C01826=1195.101,-77.193,-40.224,179.414,5.586,149.159
C01827=1195.095,-76.944,-40.234,179.416,5.586,149.159
C01828=1195.090,-76.694,-40.246,179.418,5.586,149.158
C01829=1195.084,-76.444,-40.256,179.421,5.587,149.158
C01830=1195.079,-76.194,-40.267,179.423,5.587,149.157
C01831=1195.074,-75.945,-40.278,179.425,5.587,149.156
C01832=1195.068,-75.674,-40.290,179.427,5.587,149.155
C01833=1195.063,-75.403,-40.301,179.430,5.587,149.155
C01834=1195.057,-75.133,-40.313,179.433,5.588,149.154
C01835=1195.051,-74.862,-40.325,179.435,5.588,149.153
C01836=1195.046,-74.611,-40.335,179.437,5.588,149.153
C01837=1195.041,-74.362,-40.346,179.440,5.589,149.152
C01838=1195.036,-74.112,-40.357,179.442,5.589,149.151
C01839=1195.030,-73.863,-40.368,179.444,5.589,149.151
C01840=1195.025,-73.613,-40.379,179.447,5.589,149.150
C01841=1195.020,-73.363,-40.390,179.449,5.589,149.150
C01842=1195.014,-73.113,-40.401,179.451,5.589,149.149
C01843=1195.009,-72.864,-40.412,179.454,5.590,149.148
C01844=1195.004,-72.615,-40.423,179.456,5.590,149.148
C01845=1194.999,-72.364,-40.434,179.458,5.590,149.147
C01846=1194.994,-72.115,-40.445,179.460,5.590,149.146
C01847=1194.988,-71.865,-40.455,179.463,5.590,149.146
C01848=1194.983,-71.615,-40.467,179.465,5.591,149.145
C01849=1194.977,-71.366,-40.477,179.467,5.591,149.144
C01850=1194.973,-71.116,-40.489,179.470,5.591,149.144
C01851=1194.968,-70.866,-40.499,179.473,5.592,149.143
C01852=1194.962,-70.617,-40.511,179.474,5.592,149.142
C01853=1194.957,-70.367,-40.522,179.477,5.592,149.142
C01854=1194.952,-70.117,-40.533,179.479,5.592,149.141
C01855=1194.947,-69.868,-40.544,179.482,5.592,149.140
C01856=1194.941,-69.618,-40.556,179.484,5.593,149.140
C01857=1194.936,-69.368,-40.566,179.486,5.593,149.139
C01858=1194.931,-69.119,-40.577,179.489,5.593,149.138
C01859=1194.925,-68.868,-40.588,179.491,5.593,149.138
C01860=1194.921,-68.619,-40.599,179.493,5.593,149.137
C01861=1194.915,-68.370,-40.610,179.496,5.594,149.137
C01862=1194.909,-68.119,-40.622,179.498,5.594,149.136
C01863=1194.905,-67.869,-40.633,179.500,5.594,149.135
C01864=1194.900,-67.620,-40.644,179.502,5.595,149.135
C01865=1194.895,-67.370,-40.654,179.505,5.594,149.134
C01866=1194.889,-67.120,-40.666,179.507,5.595,149.133
C01867=1194.884,-66.871,-40.677,179.510,5.595,149.133
C01868=1194.879,-66.622,-40.688,179.511,5.595,149.132
C01869=1194.873,-66.371,-40.700,179.514,5.596,149.131
C01870=1194.868,-66.122,-40.711,179.517,5.596,149.131
C01871=1194.863,-65.872,-40.722,179.519,5.596,149.130
C01872=1194.858,-65.623,-40.734,179.521,5.597,149.129
C01873=1194.853,-65.372,-40.744,179.523,5.596,149.129
C01874=1194.847,-65.123,-40.756,179.526,5.597,149.128
C01875=1194.842,-64.874,-40.767,179.529,5.597,149.127
C01876=1194.838,-64.624,-40.778,179.530,5.597,149.127
C01877=1194.831,-64.374,-40.789,179.533,5.598,149.126
C01878=1194.827,-64.125,-40.801,179.535,5.598,149.125
C01879=1194.821,-63.875,-40.812,179.538,5.598,149.125
C01880=1194.816,-63.625,-40.824,179.540,5.598,149.124
C01881=1194.811,-63.375,-40.834,179.542,5.599,149.124
C01882=1194.805,-63.125,-40.846,179.544,5.598,149.123
C01883=1194.801,-62.876,-40.857,179.547,5.599,149.122
C01884=1194.795,-62.626,-40.869,179.549,5.600,149.122
C01885=1194.790,-62.377,-40.880,179.551,5.599,149.121
C01886=1194.785,-62.127,-40.891,179.554,5.600,149.120
C01887=1194.780,-61.877,-40.902,179.557,5.600,149.120
C01888=1194.775,-61.627,-40.914,179.559,5.600,149.119
C01889=1194.769,-61.378,-40.925,179.561,5.601,149.118
C01890=1194.764,-61.128,-40.936,179.563,5.600,149.118
C01891=1194.759,-60.878,-40.948,179.566,5.601,149.117
C01892=1194.754,-60.629,-40.960,179.568,5.601,149.116
C01893=1194.749,-60.379,-40.972,179.570,5.601,149.116
C01894=1194.743,-60.130,-40.982,179.573,5.602,149.115
C01895=1194.739,-59.880,-40.994,179.575,5.602,149.114
C01896=1194.733,-59.630,-41.005,179.577,5.602,149.114
C01897=1194.728,-59.380,-41.016,179.580,5.603,149.113
C01898=1194.723,-59.130,-41.028,179.582,5.603,149.112
C01899=1194.717,-58.881,-41.039,179.584,5.603,149.112
C01900=1194.712,-58.631,-41.051,179.587,5.603,149.111
C01901=1194.707,-58.382,-41.062,179.590,5.603,149.110
C01902=1194.702,-58.132,-41.074,179.591,5.604,149.110
C01903=1194.697,-57.882,-41.085,179.594,5.604,149.109
C01904=1194.691,-57.633,-41.097,179.597,5.604,149.108
C01905=1194.686,-57.383,-41.108,179.599,5.604,149.108
C01906=1194.681,-57.133,-41.120,179.601,5.605,149.107
C01907=1194.676,-56.884,-41.131,179.604,5.605,149.107
C01908=1194.671,-56.634,-41.143,179.606,5.605,149.106
C01909=1194.665,-56.384,-41.155,179.608,5.605,149.105
C01910=1194.661,-56.134,-41.166,179.611,5.606,149.104
C01911=1194.655,-55.885,-41.178,179.613,5.606,149.104
C01912=1194.650,-55.635,-41.189,179.615,5.606,149.103
C01913=1194.645,-55.385,-41.201,179.618,5.607,149.103
C01914=1194.640,-55.136,-41.212,179.620,5.606,149.102
C01915=1194.635,-54.886,-41.224,179.622,5.607,149.101
C01916=1194.630,-54.636,-41.236,179.625,5.608,149.101
C01917=1194.624,-54.386,-41.247,179.627,5.608,149.100
C01918=1194.618,-54.137,-41.259,179.630,5.608,149.099
C01919=1194.614,-53.887,-41.270,179.632,5.609,149.099
C01920=1194.609,-53.638,-41.283,179.634,5.609,149.098
C01921=1194.604,-53.388,-41.294,179.636,5.609,149.097
C01922=1194.598,-53.139,-41.306,179.639,5.609,149.097
C01923=1194.593,-52.889,-41.318,179.642,5.609,149.096
C01924=1194.588,-52.639,-41.329,179.643,5.609,149.096
C01925=1194.583,-52.389,-41.341,179.646,5.610,149.095
C01926=1194.577,-52.139,-41.353,179.649,5.610,149.094
C01927=1194.572,-51.890,-41.364,179.651,5.610,149.093
C01928=1194.567,-51.641,-41.376,179.653,5.611,149.093
C01929=1194.562,-51.391,-41.388,179.656,5.611,149.092
C01930=1194.557,-51.141,-41.400,179.658,5.611,149.092
C01931=1194.551,-50.891,-41.412,179.660,5.611,149.091
C01932=1194.547,-50.642,-41.423,179.663,5.612,149.090
C01933=1194.541,-50.392,-41.435,179.665,5.613,149.090
C01934=1194.536,-50.142,-41.447,179.667,5.612,149.089
C01935=1194.531,-49.893,-41.459,179.670,5.613,149.088
C01936=1194.525,-49.623,-41.472,179.673,5.613,149.088
C01937=1194.520,-49.353,-41.485,179.675,5.614,149.087
C01938=1194.514,-49.082,-41.497,179.677,5.613,149.086
C01939=1194.508,-48.812,-41.510,179.680,5.614,149.085
C01940=1194.504,-48.563,-41.522,179.683,5.614,149.085
C01941=1194.498,-48.313,-41.534,179.685,5.615,149.084
C01942=1194.493,-48.063,-41.545,179.687,5.615,149.084
C01943=1194.487,-47.813,-41.557,179.690,5.615,149.083
C01944=1194.483,-47.564,-41.569,179.692,5.615,149.082
C01945=1194.478,-47.314,-41.581,179.695,5.616,149.081
C01946=1194.472,-47.064,-41.593,179.697,5.616,149.081
C01947=1194.467,-46.814,-41.605,179.699,5.616,149.080
C01948=1194.462,-46.565,-41.617,179.702,5.617,149.080
C01949=1194.457,-46.315,-41.629,179.704,5.616,149.079
C01950=1194.451,-46.065,-41.641,179.707,5.617,149.078
C01951=1194.446,-45.816,-41.653,179.709,5.618,149.078
C01952=1194.442,-45.566,-41.665,179.711,5.617,149.077
C01953=1194.436,-45.316,-41.676,179.714,5.618,149.076
C01954=1194.431,-45.067,-41.689,179.716,5.618,149.076
C01955=1194.426,-44.817,-41.701,179.719,5.619,149.075
C01956=1194.420,-44.567,-41.713,179.721,5.619,149.074
C01957=1194.416,-44.318,-41.725,179.723,5.619,149.074
C01958=1194.410,-44.068,-41.737,179.726,5.620,149.073
C01959=1194.405,-43.819,-41.749,179.729,5.620,149.072
C01960=1194.400,-43.569,-41.761,179.731,5.620,149.072
C01961=1194.394,-43.319,-41.773,179.733,5.621,149.071
C01962=1194.389,-43.070,-41.786,179.735,5.621,149.070
C01963=1194.385,-42.820,-41.797,179.738,5.621,149.070
C01964=1194.379,-42.571,-41.810,179.740,5.621,149.069
C01965=1194.374,-42.321,-41.822,179.742,5.622,149.069
C01966=1194.369,-42.071,-41.833,179.745,5.622,149.068
C01967=1194.364,-41.822,-41.846,179.747,5.622,149.067
C01968=1194.358,-41.572,-41.858,179.750,5.623,149.066
C01969=1194.354,-41.323,-41.870,179.752,5.623,149.066
C01970=1194.348,-41.073,-41.882,179.755,5.624,149.065
C01971=1194.343,-40.824,-41.894,179.757,5.623,149.065
C01972=1194.338,-40.574,-41.906,179.759,5.624,149.064
C01973=1194.333,-40.324,-41.919,179.762,5.624,149.063
C01974=1194.328,-40.074,-41.931,179.764,5.624,149.062
C01975=1194.323,-39.824,-41.944,179.766,5.625,149.062
C01976=1194.317,-39.574,-41.956,179.769,5.625,149.061
C01977=1194.312,-39.325,-41.968,179.772,5.626,149.061
C01978=1194.307,-39.075,-41.980,179.774,5.625,149.060
C01979=1194.302,-38.826,-41.992,179.776,5.626,149.059
C01980=1194.297,-38.576,-42.004,179.779,5.627,149.059
C01981=1194.292,-38.327,-42.017,179.781,5.627,149.058
C01982=1194.286,-38.077,-42.028,179.783,5.627,149.057
C01983=1194.281,-37.828,-42.041,179.786,5.627,149.057
C01984=1194.276,-37.578,-42.053,179.789,5.628,149.056
C01985=1194.271,-37.328,-42.066,179.791,5.629,149.055
C01986=1194.266,-37.078,-42.078,179.793,5.628,149.055
C01987=1194.261,-36.828,-42.090,179.796,5.629,149.054
C01988=1194.256,-36.579,-42.103,179.798,5.629,149.053
C01989=1194.250,-36.329,-42.115,179.800,5.630,149.053
C01990=1194.245,-36.080,-42.127,179.802,5.630,149.052
C01991=1194.240,-35.830,-42.139,179.805,5.630,149.051
C01992=1194.234,-35.581,-42.152,179.808,5.630,149.051
C01993=1194.229,-35.331,-42.165,179.810,5.631,149.050
C01994=1194.224,-35.081,-42.177,179.812,5.631,149.050
C01995=1194.219,-34.831,-42.189,179.815,5.631,149.049
C01996=1194.214,-34.582,-42.202,179.817,5.632,149.048
C01997=1194.209,-34.332,-42.214,179.820,5.632,149.048
C01998=1194.204,-34.083,-42.226,179.822,5.632,149.047
C01999=1194.199,-33.833,-42.239,179.824,5.633,149.046
C02000=1194.193,-33.583,-42.251,179.827,5.633,149.046
C02001=1194.189,-33.333,-42.264,179.830,5.634,149.045
C02002=1194.183,-33.084,-42.277,179.832,5.633,149.044
C02003=1194.178,-32.834,-42.288,179.834,5.634,149.044
C02004=1194.173,-32.585,-42.301,179.836,5.635,149.043
C02005=1194.168,-32.336,-42.314,179.839,5.635,149.042
C02006=1194.163,-32.086,-42.327,179.842,5.636,149.042
C02007=1194.157,-31.835,-42.339,179.844,5.635,149.041
C02008=1194.152,-31.586,-42.352,179.847,5.636,149.040
C02009=1194.147,-31.337,-42.364,179.849,5.637,149.040
C02010=1194.142,-31.087,-42.377,179.851,5.637,149.039
C02011=1194.136,-30.837,-42.389,179.853,5.637,149.038
C02012=1194.132,-30.587,-42.402,179.856,5.637,149.038
C02013=1194.127,-30.338,-42.414,179.859,5.638,149.037
C02014=1194.122,-30.089,-42.427,179.861,5.638,149.037
C02015=1194.116,-29.839,-42.440,179.863,5.638,149.036
C02016=1194.112,-29.589,-42.452,179.866,5.639,149.035
C02017=1194.106,-29.339,-42.465,179.868,5.639,149.034
C02018=1194.101,-29.090,-42.478,179.871,5.639,149.034
C02019=1194.095,-28.841,-42.490,179.873,5.640,149.033
C02020=1194.090,-28.591,-42.503,179.875,5.640,149.033
C02021=1194.086,-28.341,-42.516,179.878,5.640,149.032
C02022=1194.080,-28.091,-42.528,179.881,5.641,149.031
C02023=1194.075,-27.842,-42.540,179.883,5.641,149.031
C02024=1194.069,-27.592,-42.553,179.885,5.642,149.030
C02025=1194.065,-27.342,-42.566,179.888,5.642,149.029
C02026=1194.060,-27.093,-42.579,179.890,5.642,149.029
C02027=1194.055,-26.844,-42.592,179.893,5.643,149.028
C02028=1194.050,-26.594,-42.604,179.895,5.644,149.027
C02029=1194.045,-26.344,-42.617,179.897,5.643,149.027
C02030=1194.039,-26.094,-42.630,179.900,5.644,149.026
C02031=1194.034,-25.845,-42.642,179.902,5.644,149.025
C02032=1194.029,-25.595,-42.655,179.905,5.645,149.025
C02033=1194.024,-25.345,-42.668,179.907,5.645,149.024
C02034=1194.019,-25.096,-42.680,179.909,5.645,149.024
C02035=1194.013,-24.846,-42.694,179.912,5.646,149.023
C02036=1194.009,-24.596,-42.707,179.915,5.646,149.022
C02037=1194.003,-24.347,-42.719,179.917,5.647,149.021
C02038=1193.998,-24.098,-42.732,179.919,5.647,149.021
C02039=1193.993,-23.847,-42.745,179.922,5.647,149.020
C02040=1193.987,-23.578,-42.759,179.924,5.648,149.020
C02041=1193.982,-23.309,-42.772,179.927,5.648,149.019
C02042=1193.977,-23.039,-42.787,179.930,5.648,149.018
C02043=1193.971,-22.770,-42.800,179.932,5.649,149.018
C02044=1193.966,-22.519,-42.813,179.935,5.649,149.017
C02045=1193.961,-22.270,-42.826,179.938,5.650,149.016
C02046=1193.956,-22.021,-42.839,179.940,5.650,149.015
C02047=1193.950,-21.770,-42.852,179.942,5.650,149.015
C02048=1193.946,-21.522,-42.866,179.944,5.651,149.014
C02049=1193.940,-21.272,-42.878,179.947,5.651,149.014
C02050=1193.935,-21.022,-42.892,179.950,5.652,149.013
C02051=1193.930,-20.773,-42.904,179.952,5.652,149.012
C02052=1193.925,-20.523,-42.917,179.955,5.653,149.012
C02053=1193.920,-20.273,-42.931,179.957,5.653,149.011
C02054=1193.914,-20.024,-42.943,179.959,5.653,149.010
C02055=1193.909,-19.774,-42.956,179.962,5.654,149.010
C02056=1193.904,-19.524,-42.969,179.965,5.654,149.009
C02057=1193.899,-19.275,-42.982,179.967,5.655,149.008
C02058=1193.894,-19.025,-42.995,179.969,5.655,149.008
C02059=1193.889,-18.776,-43.009,179.972,5.655,149.007
C02060=1193.884,-18.526,-43.021,179.974,5.656,149.006
C02061=1193.879,-18.276,-43.034,179.977,5.656,149.006
C02062=1193.873,-18.027,-43.048,179.979,5.657,149.005
C02063=1193.868,-17.777,-43.060,179.982,5.657,149.005
C02064=1193.863,-17.527,-43.074,179.984,5.657,149.004
C02065=1193.858,-17.278,-43.087,179.986,5.657,149.003
C02066=1193.854,-17.028,-43.100,179.989,5.658,149.002
C02067=1193.848,-16.779,-43.113,179.991,5.659,149.002
C02068=1193.843,-16.529,-43.126,179.994,5.659,149.001
C02069=1193.837,-16.279,-43.139,179.997,5.660,149.001
C02070=1193.833,-16.030,-43.153,179.999,5.659,149.000
C02071=1193.828,-15.780,-43.166,-179.999,5.660,148.999
C02072=1193.822,-15.531,-43.179,-179.997,5.661,148.999
C02073=1193.818,-15.281,-43.192,-179.994,5.661,148.998
C02074=1193.812,-15.032,-43.206,-179.991,5.662,148.997
C02075=1193.807,-14.782,-43.218,-179.989,5.662,148.997
C02076=1193.802,-14.532,-43.232,-179.986,5.663,148.996
C02077=1193.797,-14.283,-43.244,-179.984,5.663,148.995
C02078=1193.792,-14.033,-43.259,-179.982,5.663,148.995
C02079=1193.787,-13.784,-43.271,-179.979,5.664,148.994
C02080=1193.782,-13.534,-43.284,-179.976,5.664,148.993
C02081=1193.776,-13.285,-43.298,-179.974,5.665,148.993
C02082=1193.772,-13.035,-43.311,-179.972,5.665,148.992
C02083=1193.766,-12.785,-43.324,-179.969,5.665,148.992
C02084=1193.762,-12.536,-43.338,-179.967,5.666,148.991
C02085=1193.756,-12.286,-43.351,-179.964,5.666,148.990
C02086=1193.751,-12.037,-43.364,-179.962,5.667,148.990
C02087=1193.746,-11.787,-43.378,-179.959,5.667,148.989
C02088=1193.741,-11.538,-43.391,-179.957,5.668,148.988
C02089=1193.736,-11.287,-43.404,-179.954,5.668,148.988
C02090=1193.730,-11.038,-43.418,-179.952,5.668,148.987
C02091=1193.725,-10.788,-43.431,-179.950,5.669,148.986
C02092=1193.720,-10.539,-43.445,-179.947,5.669,148.986
C02093=1193.715,-10.289,-43.458,-179.944,5.670,148.985
C02094=1193.710,-10.040,-43.471,-179.942,5.670,148.984
C02095=1193.705,-9.790,-43.485,-179.939,5.671,148.984
C02096=1193.699,-9.541,-43.498,-179.937,5.672,148.983
C02097=1193.695,-9.291,-43.512,-179.935,5.671,148.983
C02098=1193.690,-9.041,-43.525,-179.932,5.672,148.982
C02099=1193.685,-8.792,-43.539,-179.930,5.672,148.981
C02100=1193.680,-8.542,-43.552,-179.927,5.673,148.980
C02101=1193.674,-8.293,-43.566,-179.925,5.674,148.980
C02102=1193.670,-8.043,-43.579,-179.922,5.674,148.979
C02103=1193.664,-7.794,-43.593,-179.919,5.674,148.979
C02104=1193.660,-7.544,-43.606,-179.917,5.675,148.978
C02105=1193.654,-7.295,-43.620,-179.915,5.675,148.977
C02106=1193.649,-7.045,-43.633,-179.913,5.675,148.977
C02107=1193.644,-6.796,-43.647,-179.910,5.676,148.976
C02108=1193.639,-6.546,-43.660,-179.907,5.676,148.975
C02109=1193.634,-6.296,-43.675,-179.905,5.677,148.975
C02110=1193.629,-6.046,-43.687,-179.902,5.678,148.974
C02111=1193.624,-5.797,-43.701,-179.900,5.678,148.974
C02112=1193.618,-5.547,-43.715,-179.897,5.679,148.973
C02113=1193.614,-5.298,-43.728,-179.894,5.679,148.972
C02114=1193.608,-5.048,-43.742,-179.892,5.679,148.971
C02115=1193.603,-4.798,-43.756,-179.890,5.680,148.971
C02116=1193.599,-4.549,-43.770,-179.888,5.680,148.970
C02117=1193.593,-4.299,-43.783,-179.885,5.681,148.970
C02118=1193.588,-4.050,-43.797,-179.882,5.681,148.969
C02119=1193.583,-3.800,-43.810,-179.880,5.682,148.969
C02120=1193.578,-3.551,-43.824,-179.877,5.682,148.968
C02121=1193.573,-3.301,-43.838,-179.875,5.683,148.967
C02122=1193.568,-3.052,-43.851,-179.872,5.683,148.966
C02123=1193.563,-2.802,-43.865,-179.870,5.683,148.966
C02124=1193.557,-2.553,-43.879,-179.868,5.684,148.965
C02125=1193.552,-2.303,-43.892,-179.865,5.684,148.965
C02126=1193.548,-2.053,-43.906,-179.863,5.685,148.964
C02127=1193.542,-1.804,-43.920,-179.860,5.685,148.963
C02128=1193.537,-1.554,-43.934,-179.857,5.686,148.963
C02129=1193.532,-1.304,-43.948,-179.855,5.687,148.962
C02130=1193.527,-1.055,-43.961,-179.852,5.687,148.961
C02131=1193.522,-0.805,-43.975,-179.850,5.688,148.961
C02132=1193.517,-0.555,-43.989,-179.847,5.688,148.960
C02133=1193.511,-0.306,-44.003,-179.845,5.689,148.960
C02134=1193.507,-0.057,-44.017,-179.843,5.689,148.959
C02135=1193.502,0.193,-44.030,-179.840,5.689,148.958
C02136=1193.496,0.442,-44.044,-179.838,5.690,148.957
C02137=1193.491,0.692,-44.058,-179.835,5.690,148.957
C02138=1193.486,0.942,-44.073,-179.833,5.691,148.956
C02139=1193.481,1.191,-44.085,-179.830,5.692,148.956
C02140=1193.476,1.441,-44.100,-179.827,5.692,148.955
C02141=1193.471,1.691,-44.114,-179.825,5.693,148.954
C02142=1193.466,1.940,-44.128,-179.823,5.693,148.954
C02143=1193.461,2.189,-44.142,-179.820,5.694,148.953
C02144=1193.455,2.459,-44.157,-179.817,5.694,148.952
C02145=1193.450,2.728,-44.172,-179.815,5.695,148.952
C02146=1193.444,2.997,-44.187,-179.812,5.695,148.951
C02147=1193.439,3.266,-44.202,-179.809,5.696,148.950
C02148=1193.434,3.516,-44.215,-179.807,5.696,148.950
C02149=1193.429,3.765,-44.230,-179.804,5.697,148.949
C02150=1193.424,4.014,-44.244,-179.801,5.697,148.948
C02151=1193.419,4.264,-44.258,-179.799,5.698,148.948
C02152=1193.414,4.514,-44.272,-179.797,5.699,148.947
C02153=1193.408,4.763,-44.286,-179.794,5.699,148.946
C02154=1193.403,5.012,-44.300,-179.792,5.699,148.946
C02155=1193.398,5.262,-44.315,-179.790,5.700,148.945
C02156=1193.393,5.513,-44.328,-179.787,5.700,148.945
C02157=1193.388,5.761,-44.341,-179.784,5.701,148.944
C02158=1193.383,6.011,-44.356,-179.782,5.701,148.943
C02159=1193.378,6.261,-44.370,-179.779,5.702,148.943
C02160=1193.374,6.510,-44.384,-179.777,5.702,148.942
C02161=1193.368,6.759,-44.398,-179.774,5.703,148.941
C02162=1193.363,7.009,-44.412,-179.772,5.703,148.941
C02163=1193.358,7.259,-44.427,-179.769,5.704,148.940
C02164=1193.353,7.508,-44.441,-179.767,5.705,148.940
C02165=1193.348,7.758,-44.455,-179.764,5.705,148.939
C02166=1193.343,8.007,-44.469,-179.761,5.706,148.938
C02167=1193.338,8.257,-44.483,-179.759,5.706,148.938
C02168=1193.333,8.507,-44.498,-179.757,5.707,148.937
C02169=1193.328,8.756,-44.512,-179.754,5.708,148.936
C02170=1193.322,9.005,-44.526,-179.751,5.708,148.936
C02171=1193.317,9.255,-44.540,-179.749,5.709,148.935
C02172=1193.312,9.505,-44.554,-179.746,5.709,148.934
C02173=1193.307,9.754,-44.569,-179.744,5.709,148.934
C02174=1193.302,10.004,-44.583,-179.742,5.710,148.933
C02175=1193.297,10.254,-44.597,-179.739,5.710,148.933
C02176=1193.292,10.502,-44.612,-179.737,5.711,148.932
C02177=1193.287,10.752,-44.626,-179.734,5.712,148.931
C02178=1193.282,11.002,-44.640,-179.732,5.712,148.931
C02179=1193.277,11.251,-44.655,-179.729,5.712,148.930
C02180=1193.272,11.501,-44.669,-179.726,5.713,148.929
C02181=1193.267,11.750,-44.683,-179.724,5.714,148.929
C02182=1193.262,12.000,-44.697,-179.722,5.714,148.928
C02183=1193.257,12.250,-44.712,-179.719,5.715,148.927
C02184=1193.252,12.499,-44.726,-179.716,5.715,148.927
C02185=1193.247,12.748,-44.741,-179.714,5.716,148.926
C02186=1193.242,12.998,-44.755,-179.711,5.717,148.926
C02187=1193.237,13.248,-44.769,-179.709,5.717,148.925
C02188=1193.231,13.497,-44.784,-179.706,5.718,148.924
C02189=1193.226,13.747,-44.798,-179.704,5.718,148.924
C02190=1193.221,13.997,-44.812,-179.701,5.719,148.923
C02191=1193.216,14.246,-44.827,-179.699,5.720,148.922
C02192=1193.212,14.495,-44.842,-179.696,5.720,148.922
C02193=1193.207,14.745,-44.856,-179.693,5.721,148.921
C02194=1193.202,14.995,-44.870,-179.691,5.721,148.921
C02195=1193.197,15.244,-44.885,-179.689,5.722,148.920
C02196=1193.191,15.493,-44.900,-179.686,5.722,148.919
C02197=1193.186,15.743,-44.914,-179.683,5.723,148.919
C02198=1193.181,15.993,-44.928,-179.681,5.724,148.918
C02199=1193.176,16.242,-44.943,-179.679,5.724,148.917
C02200=1193.171,16.491,-44.958,-179.676,5.725,148.917
C02201=1193.166,16.741,-44.972,-179.673,5.725,148.916
C02202=1193.161,16.990,-44.987,-179.671,5.726,148.916
C02203=1193.156,17.240,-45.002,-179.668,5.727,148.915
C02204=1193.151,17.490,-45.016,-179.666,5.727,148.914
C02205=1193.146,17.740,-45.030,-179.663,5.728,148.914
C02206=1193.141,17.989,-45.045,-179.661,5.728,148.913
C02207=1193.136,18.238,-45.060,-179.658,5.729,148.912
C02208=1193.131,18.488,-45.074,-179.656,5.729,148.912
C02209=1193.126,18.738,-45.089,-179.653,5.730,148.911
C02210=1193.120,18.987,-45.103,-179.651,5.731,148.911
C02211=1193.116,19.236,-45.118,-179.648,5.731,148.910
C02212=1193.110,19.486,-45.133,-179.646,5.732,148.909
C02213=1193.105,19.735,-45.147,-179.643,5.732,148.909
C02214=1193.101,19.984,-45.162,-179.641,5.733,148.908
C02215=1193.096,20.234,-45.177,-179.638,5.734,148.907
C02216=1193.090,20.484,-45.192,-179.635,5.734,148.907
C02217=1193.085,20.733,-45.207,-179.633,5.735,148.906
C02218=1193.080,20.983,-45.221,-179.631,5.736,148.906
C02219=1193.076,21.232,-45.236,-179.628,5.736,148.905
C02220=1193.070,21.482,-45.251,-179.625,5.737,148.904
C02221=1193.065,21.731,-45.266,-179.623,5.737,148.904
C02222=1193.060,21.981,-45.280,-179.621,5.738,148.903
C02223=1193.055,22.230,-45.296,-179.618,5.738,148.902
C02224=1193.050,22.480,-45.310,-179.615,5.739,148.902
C02225=1193.045,22.729,-45.325,-179.613,5.739,148.901
C02226=1193.040,22.979,-45.339,-179.610,5.740,148.901
C02227=1193.035,23.228,-45.355,-179.608,5.741,148.900
C02228=1193.030,23.478,-45.369,-179.605,5.741,148.899
C02229=1193.025,23.727,-45.384,-179.602,5.742,148.899
C02230=1193.020,23.977,-45.399,-179.600,5.743,148.898
C02231=1193.015,24.226,-45.414,-179.598,5.743,148.897
C02232=1193.010,24.476,-45.428,-179.595,5.744,148.897
C02233=1193.005,24.725,-45.444,-179.592,5.744,148.896
C02234=1193.000,24.975,-45.458,-179.590,5.745,148.896
C02235=1192.994,25.224,-45.474,-179.588,5.746,148.895
C02236=1192.990,25.474,-45.489,-179.585,5.746,148.894
C02237=1192.985,25.724,-45.503,-179.583,5.747,148.894
C02238=1192.980,25.973,-45.519,-179.580,5.748,148.893
C02239=1192.975,26.223,-45.533,-179.577,5.748,148.893
C02240=1192.970,26.472,-45.549,-179.574,5.749,148.892
C02241=1192.965,26.721,-45.564,-179.572,5.750,148.891
C02242=1192.960,26.971,-45.578,-179.569,5.751,148.891
C02243=1192.955,27.221,-45.594,-179.567,5.751,148.890
C02244=1192.950,27.470,-45.608,-179.564,5.752,148.889
C02245=1192.944,27.720,-45.623,-179.562,5.753,148.889
C02246=1192.940,27.969,-45.638,-179.559,5.753,148.888
C02247=1192.935,28.218,-45.653,-179.557,5.754,148.888
C02248=1192.929,28.487,-45.670,-179.554,5.754,148.887
C02249=1192.923,28.756,-45.686,-179.551,5.755,148.886
C02250=1192.918,29.025,-45.702,-179.548,5.756,148.886
C02251=1192.913,29.293,-45.719,-179.546,5.756,148.885
C02252=1192.908,29.542,-45.734,-179.543,5.757,148.884
C02253=1192.903,29.793,-45.749,-179.541,5.758,148.884
C02254=1192.898,30.042,-45.764,-179.538,5.758,148.883
C02255=1192.893,30.292,-45.779,-179.536,5.759,148.883
C02256=1192.888,30.541,-45.794,-179.533,5.760,148.882
C02257=1192.882,30.791,-45.809,-179.531,5.760,148.881
C02258=1192.878,31.040,-45.824,-179.528,5.761,148.881
C02259=1192.872,31.289,-45.840,-179.526,5.762,148.880
C02260=1192.868,31.539,-45.855,-179.523,5.762,148.879
C02261=1192.863,31.789,-45.870,-179.521,5.763,148.879
C02262=1192.858,32.038,-45.885,-179.518,5.763,148.878
C02263=1192.853,32.288,-45.901,-179.515,5.765,148.878
C02264=1192.848,32.537,-45.916,-179.513,5.765,148.877
C02265=1192.843,32.786,-45.931,-179.510,5.766,148.876
C02266=1192.838,33.036,-45.946,-179.508,5.767,148.876
C02267=1192.833,33.286,-45.962,-179.505,5.767,148.875
C02268=1192.828,33.535,-45.977,-179.502,5.768,148.874
C02269=1192.823,33.784,-45.992,-179.500,5.768,148.874
C02270=1192.817,34.034,-46.008,-179.498,5.769,148.873
C02271=1192.813,34.283,-46.023,-179.495,5.770,148.873
C02272=1192.808,34.533,-46.039,-179.492,5.770,148.872
C02273=1192.803,34.782,-46.054,-179.490,5.771,148.872
C02274=1192.798,35.031,-46.069,-179.488,5.772,148.871
C02275=1192.792,35.281,-46.084,-179.484,5.773,148.870
C02276=1192.788,35.531,-46.099,-179.482,5.773,148.870
C02277=1192.783,35.781,-46.115,-179.480,5.774,148.869
C02278=1192.778,36.030,-46.130,-179.477,5.775,148.868
C02279=1192.773,36.279,-46.146,-179.474,5.775,148.868
C02280=1192.767,36.529,-46.161,-179.472,5.776,148.867
C02281=1192.763,36.778,-46.177,-179.469,5.777,148.867
C02282=1192.758,37.028,-46.192,-179.467,5.777,148.866
C02283=1192.753,37.277,-46.208,-179.464,5.778,148.865
C02284=1192.748,37.526,-46.223,-179.462,5.779,148.865
C02285=1192.743,37.776,-46.238,-179.459,5.779,148.864
C02286=1192.738,38.026,-46.254,-179.456,5.780,148.863
C02287=1192.733,38.275,-46.269,-179.454,5.781,148.863
C02288=1192.728,38.524,-46.285,-179.451,5.782,148.862
C02289=1192.722,38.774,-46.300,-179.449,5.782,148.862
C02290=1192.718,39.024,-46.316,-179.447,5.783,148.861
C02291=1192.713,39.273,-46.331,-179.444,5.784,148.861
C02292=1192.708,39.522,-46.347,-179.441,5.784,148.860
C02293=1192.703,39.772,-46.363,-179.439,5.785,148.859
C02294=1192.698,40.021,-46.378,-179.436,5.786,148.859
C02295=1192.693,40.270,-46.394,-179.433,5.787,148.858
C02296=1192.688,40.520,-46.410,-179.431,5.788,148.857
C02297=1192.683,40.770,-46.426,-179.428,5.788,148.857
C02298=1192.678,41.019,-46.441,-179.426,5.789,148.856
C02299=1192.673,41.268,-46.456,-179.423,5.789,148.856
C02300=1192.668,41.518,-46.472,-179.421,5.790,148.855
C02301=1192.663,41.768,-46.488,-179.418,5.791,148.855
C02302=1192.658,42.017,-46.503,-179.416,5.791,148.854
C02303=1192.654,42.266,-46.520,-179.413,5.793,148.853
C02304=1192.648,42.516,-46.535,-179.410,5.794,148.853
C02305=1192.643,42.765,-46.551,-179.408,5.794,148.852
C02306=1192.637,43.015,-46.566,-179.405,5.795,148.851
C02307=1192.633,43.264,-46.582,-179.403,5.796,148.851
C02308=1192.628,43.513,-46.598,-179.400,5.796,148.850
C02309=1192.623,43.763,-46.614,-179.398,5.797,148.850
C02310=1192.618,44.013,-46.630,-179.396,5.797,148.849
C02311=1192.613,44.262,-46.645,-179.392,5.799,148.848
C02312=1192.608,44.512,-46.661,-179.390,5.799,148.848
C02313=1192.604,44.761,-46.677,-179.388,5.800,148.847
C02314=1192.598,45.010,-46.692,-179.385,5.801,148.847
C02315=1192.593,45.260,-46.708,-179.382,5.801,148.846
C02316=1192.588,45.510,-46.724,-179.380,5.802,148.846
C02317=1192.583,45.758,-46.740,-179.377,5.803,148.845
C02318=1192.578,46.008,-46.756,-179.374,5.804,148.844
C02319=1192.573,46.258,-46.772,-179.372,5.805,148.844
C02320=1192.569,46.507,-46.788,-179.369,5.805,148.843
C02321=1192.564,46.756,-46.803,-179.367,5.806,148.842
C02322=1192.558,47.006,-46.819,-179.364,5.806,148.842
C02323=1192.554,47.255,-46.836,-179.362,5.807,148.841
C02324=1192.548,47.505,-46.851,-179.359,5.809,148.841
C02325=1192.544,47.755,-46.867,-179.356,5.809,148.840
C02326=1192.538,48.004,-46.884,-179.354,5.810,148.840
C02327=1192.533,48.253,-46.899,-179.351,5.811,148.839
C02328=1192.528,48.503,-46.915,-179.349,5.811,148.838
C02329=1192.523,48.752,-46.931,-179.347,5.812,148.838
C02330=1192.518,49.002,-46.947,-179.343,5.813,148.837
C02331=1192.513,49.251,-46.964,-179.341,5.814,148.836
C02332=1192.508,49.500,-46.979,-179.339,5.815,148.836
C02333=1192.503,49.750,-46.995,-179.336,5.815,148.835
C02334=1192.499,49.999,-47.011,-179.333,5.816,148.835
C02335=1192.494,50.249,-47.027,-179.331,5.817,148.834
C02336=1192.489,50.498,-47.043,-179.328,5.818,148.834
C02337=1192.484,50.748,-47.059,-179.325,5.819,148.833
C02338=1192.479,50.996,-47.075,-179.323,5.819,148.832
C02339=1192.474,51.247,-47.091,-179.320,5.820,148.832
C02340=1192.469,51.495,-47.108,-179.318,5.821,148.831
C02341=1192.464,51.745,-47.124,-179.316,5.821,148.831
C02342=1192.459,51.994,-47.140,-179.312,5.823,148.830
C02343=1192.455,52.244,-47.156,-179.310,5.823,148.829
C02344=1192.450,52.493,-47.172,-179.308,5.824,148.829
C02345=1192.444,52.744,-47.189,-179.305,5.825,148.828
C02346=1192.439,52.992,-47.205,-179.302,5.825,148.828
C02347=1192.434,53.242,-47.221,-179.300,5.827,148.827
C02348=1192.429,53.491,-47.237,-179.297,5.827,148.826
C02349=1192.425,53.741,-47.254,-179.294,5.828,148.826
C02350=1192.419,53.990,-47.270,-179.292,5.829,148.825
C02351=1192.415,54.240,-47.286,-179.290,5.829,148.825
C02352=1192.409,54.508,-47.303,-179.286,5.831,148.824
C02353=1192.404,54.777,-47.320,-179.284,5.831,148.823
C02354=1192.399,55.045,-47.338,-179.282,5.832,148.823
C02355=1192.393,55.314,-47.356,-179.278,5.834,148.822
C02356=1192.388,55.563,-47.372,-179.276,5.834,148.822
C02357=1192.383,55.812,-47.389,-179.273,5.835,148.821
C02358=1192.378,56.062,-47.405,-179.271,5.835,148.820
C02359=1192.373,56.311,-47.421,-179.268,5.837,148.820
C02360=1192.368,56.561,-47.437,-179.265,5.837,148.819
C02361=1192.363,56.810,-47.453,-179.263,5.838,148.819
C02362=1192.359,57.059,-47.470,-179.260,5.839,148.818
C02363=1192.353,57.309,-47.487,-179.258,5.840,148.818
C02364=1192.348,57.559,-47.503,-179.255,5.841,148.817
C02365=1192.343,57.807,-47.519,-179.252,5.842,148.816
C02366=1192.339,58.057,-47.536,-179.250,5.842,148.816
C02367=1192.333,58.306,-47.552,-179.248,5.843,148.815
C02368=1192.329,58.556,-47.568,-179.245,5.844,148.815
C02369=1192.324,58.806,-47.585,-179.242,5.845,148.814
C02370=1192.319,59.054,-47.602,-179.240,5.846,148.813
C02371=1192.314,59.304,-47.618,-179.237,5.846,148.813
C02372=1192.309,59.553,-47.634,-179.235,5.847,148.812
C02373=1192.304,59.803,-47.651,-179.232,5.849,148.812
C02374=1192.299,60.053,-47.668,-179.229,5.849,148.811
C02375=1192.294,60.301,-47.684,-179.227,5.850,148.811
C02376=1192.289,60.551,-47.700,-179.224,5.850,148.810
C02377=1192.284,60.800,-47.717,-179.222,5.851,148.809
C02378=1192.279,61.050,-47.734,-179.219,5.853,148.809
C02379=1192.274,61.299,-47.750,-179.216,5.853,148.808
C02380=1192.269,61.548,-47.767,-179.214,5.854,148.808
C02381=1192.265,61.798,-47.783,-179.211,5.855,148.807
C02382=1192.259,62.048,-47.800,-179.208,5.856,148.806
C02383=1192.254,62.297,-47.816,-179.206,5.857,148.806
C02384=1192.250,62.546,-47.833,-179.203,5.857,148.805
C02385=1192.244,62.796,-47.850,-179.201,5.858,148.805
C02386=1192.239,63.045,-47.867,-179.198,5.860,148.804
C02387=1192.235,63.294,-47.883,-179.195,5.860,148.804
C02388=1192.230,63.544,-47.900,-179.193,5.861,148.803
C02389=1192.225,63.793,-47.917,-179.191,5.862,148.802
C02390=1192.220,64.043,-47.933,-179.187,5.863,148.802
C02391=1192.216,64.292,-47.950,-179.185,5.864,148.801
C02392=1192.210,64.541,-47.967,-179.183,5.864,148.801
C02393=1192.205,64.791,-47.984,-179.181,5.865,148.800
C02394=1192.201,65.040,-48.000,-179.177,5.867,148.800
C02395=1192.195,65.289,-48.017,-179.175,5.867,148.799
C02396=1192.190,65.539,-48.033,-179.173,5.868,148.798
C02397=1192.185,65.789,-48.050,-179.170,5.869,148.798
C02398=1192.180,66.037,-48.067,-179.167,5.870,148.797
C02399=1192.176,66.287,-48.084,-179.165,5.871,148.797
C02400=1192.171,66.537,-48.101,-179.162,5.872,148.796
C02401=1192.166,66.786,-48.118,-179.160,5.872,148.796
C02402=1192.161,67.035,-48.134,-179.157,5.874,148.795
C02403=1192.156,67.285,-48.152,-179.154,5.875,148.795
C02404=1192.151,67.534,-48.168,-179.152,5.875,148.794
C02405=1192.145,67.783,-48.185,-179.149,5.877,148.793
C02406=1192.141,68.033,-48.202,-179.146,5.877,148.793
C02407=1192.136,68.282,-48.219,-179.144,5.878,148.792
C02408=1192.131,68.532,-48.236,-179.142,5.879,148.792
C02409=1192.126,68.781,-48.252,-179.138,5.880,148.791
C02410=1192.121,69.030,-48.269,-179.136,5.881,148.790
C02411=1192.117,69.280,-48.286,-179.134,5.882,148.790
C02412=1192.112,69.529,-48.304,-179.131,5.882,148.789
C02413=1192.107,69.779,-48.321,-179.128,5.884,148.789
C02414=1192.101,70.028,-48.338,-179.126,5.885,148.788
C02415=1192.097,70.277,-48.354,-179.123,5.885,148.788
C02416=1192.092,70.527,-48.372,-179.120,5.887,148.787
C02417=1192.087,70.777,-48.388,-179.118,5.887,148.786
C02418=1192.082,71.025,-48.406,-179.116,5.888,148.786
C02419=1192.077,71.274,-48.422,-179.113,5.889,148.785
C02420=1192.072,71.524,-48.440,-179.110,5.890,148.785
C02421=1192.067,71.774,-48.456,-179.108,5.891,148.784
C02422=1192.063,72.023,-48.474,-179.105,5.892,148.784
C02423=1192.057,72.272,-48.491,-179.102,5.893,148.783
C02424=1192.052,72.521,-48.508,-179.100,5.894,148.783
C02425=1192.048,72.771,-48.525,-179.097,5.894,148.782
C02426=1192.043,73.020,-48.543,-179.094,5.896,148.781
C02427=1192.038,73.270,-48.559,-179.092,5.897,148.781
C02428=1192.033,73.519,-48.577,-179.089,5.898,148.780
C02429=1192.027,73.769,-48.593,-179.087,5.898,148.780
C02430=1192.023,74.017,-48.611,-179.084,5.900,148.779
C02431=1192.018,74.267,-48.628,-179.081,5.900,148.779
C02432=1192.013,74.517,-48.645,-179.079,5.901,148.778
C02433=1192.009,74.766,-48.663,-179.076,5.903,148.778
C02434=1192.003,75.016,-48.680,-179.074,5.903,148.777
C02435=1191.998,75.264,-48.696,-179.071,5.904,148.776
C02436=1191.993,75.514,-48.714,-179.068,5.905,148.776
C02437=1191.989,75.763,-48.731,-179.066,5.906,148.775
C02438=1191.984,76.013,-48.748,-179.063,5.907,148.775
C02439=1191.979,76.262,-48.766,-179.060,5.908,148.774
C02440=1191.974,76.512,-48.783,-179.058,5.909,148.774
C02441=1191.969,76.761,-48.801,-179.055,5.910,148.773
C02442=1191.964,77.011,-48.818,-179.053,5.911,148.773
C02443=1191.959,77.259,-48.834,-179.050,5.912,148.772
C02444=1191.954,77.508,-48.852,-179.048,5.913,148.771
C02445=1191.949,77.758,-48.870,-179.045,5.914,148.771
C02446=1191.945,78.007,-48.887,-179.042,5.915,148.770
C02447=1191.940,78.257,-48.904,-179.040,5.916,148.770
C02448=1191.935,78.506,-48.922,-179.037,5.917,148.769
C02449=1191.930,78.756,-48.939,-179.035,5.918,148.769
C02450=1191.925,79.005,-48.957,-179.032,5.919,148.768
C02451=1191.920,79.255,-48.974,-179.029,5.920,148.768
C02452=1191.915,79.504,-48.992,-179.027,5.921,148.767
C02453=1191.911,79.753,-49.009,-179.024,5.921,148.766
C02454=1191.906,80.002,-49.027,-179.021,5.923,148.766
C02455=1191.900,80.251,-49.044,-179.019,5.924,148.765
C02456=1191.895,80.520,-49.063,-179.017,5.925,148.765
C02457=1191.890,80.788,-49.081,-179.013,5.926,148.764
C02458=1191.885,81.057,-49.101,-179.010,5.927,148.763
C02459=1191.880,81.325,-49.119,-179.008,5.928,148.763
C02460=1191.875,81.575,-49.137,-179.005,5.929,148.762
C02461=1191.869,81.824,-49.154,-179.002,5.930,148.762
C02462=1191.865,82.073,-49.172,-179.000,5.931,148.761
C02463=1191.860,82.322,-49.189,-178.997,5.932,148.761
C02464=1191.855,82.572,-49.207,-178.995,5.933,148.760
C02465=1191.850,82.821,-49.225,-178.992,5.934,148.760
C02466=1191.844,83.070,-49.242,-178.989,5.936,148.759
C02467=1191.840,83.319,-49.259,-178.987,5.936,148.758
C02468=1191.835,83.569,-49.277,-178.985,5.937,148.758
C02469=1191.830,83.818,-49.295,-178.981,5.938,148.757
C02470=1191.825,84.067,-49.313,-178.979,5.939,148.757
C02471=1191.820,84.317,-49.331,-178.977,5.940,148.756
C02472=1191.815,84.566,-49.348,-178.973,5.941,148.756
C02473=1191.811,84.815,-49.365,-178.971,5.942,148.755
C02474=1191.806,85.065,-49.383,-178.968,5.943,148.755
C02475=1191.801,85.314,-49.401,-178.966,5.944,148.754
C02476=1191.797,85.564,-49.419,-178.963,5.945,148.754
C02477=1191.792,85.813,-49.437,-178.961,5.947,148.753
C02478=1191.787,86.063,-49.455,-178.958,5.947,148.752
C02479=1191.782,86.312,-49.473,-178.956,5.948,148.752
C02480=1191.777,86.562,-49.490,-178.953,5.950,148.751
C02481=1191.772,86.811,-49.508,-178.951,5.950,148.751
C02482=1191.767,87.060,-49.525,-178.947,5.952,148.750
C02483=1191.763,87.309,-49.543,-178.945,5.953,148.750
C02484=1191.758,87.558,-49.561,-178.943,5.953,148.749
C02485=1191.752,87.808,-49.579,-178.940,5.955,148.749
C02486=1191.748,88.057,-49.597,-178.937,5.956,148.748
C02487=1191.743,88.306,-49.615,-178.934,5.957,148.748
C02488=1191.738,88.555,-49.633,-178.932,5.958,148.747
C02489=1191.733,88.804,-49.651,-178.929,5.958,148.746
C02490=1191.728,89.054,-49.669,-178.927,5.960,148.746
C02491=1191.723,89.303,-49.686,-178.924,5.961,148.745
C02492=1191.718,89.553,-49.704,-178.921,5.962,148.745
C02493=1191.713,89.802,-49.722,-178.919,5.963,148.744
C02494=1191.709,90.052,-49.740,-178.916,5.964,148.744
C02495=1191.704,90.301,-49.758,-178.913,5.965,148.743
C02496=1191.699,90.550,-49.776,-178.911,5.966,148.743
C02497=1191.694,90.799,-49.794,-178.908,5.968,148.742
C02498=1191.689,91.048,-49.812,-178.906,5.968,148.742
C02499=1191.684,91.297,-49.830,-178.903,5.969,148.741
C02500=1191.680,91.547,-49.848,-178.900,5.971,148.741
C02501=1191.675,91.797,-49.866,-178.898,5.971,148.740
C02502=1191.670,92.046,-49.884,-178.895,5.973,148.740
C02503=1191.665,92.295,-49.902,-178.892,5.974,148.739
C02504=1191.660,92.544,-49.920,-178.890,5.975,148.739
C02505=1191.655,92.793,-49.938,-178.887,5.976,148.738
C02506=1191.650,93.042,-49.956,-178.885,5.977,148.738
C02507=1191.645,93.293,-49.975,-178.882,5.978,148.737
C02508=1191.640,93.542,-49.993,-178.880,5.979,148.736
C02509=1191.635,93.791,-50.011,-178.876,5.981,148.736
C02510=1191.630,94.040,-50.029,-178.874,5.981,148.735
C02511=1191.625,94.289,-50.047,-178.872,5.982,148.735
C02512=1191.621,94.538,-50.065,-178.869,5.984,148.734
C02513=1191.616,94.788,-50.083,-178.867,5.985,148.734
C02514=1191.611,95.038,-50.101,-178.864,5.986,148.733
C02515=1191.606,95.287,-50.119,-178.862,5.987,148.733
C02516=1191.601,95.536,-50.139,-178.858,5.988,148.732
C02517=1191.596,95.785,-50.157,-178.856,5.989,148.732
C02518=1191.592,96.035,-50.175,-178.854,5.990,148.731
C02519=1191.587,96.284,-50.193,-178.851,5.992,148.731
C02520=1191.582,96.533,-50.211,-178.848,5.992,148.730
C02521=1191.577,96.782,-50.229,-178.846,5.994,148.730
C02522=1191.572,97.032,-50.248,-178.843,5.994,148.729
C02523=1191.567,97.281,-50.267,-178.840,5.996,148.729
C02524=1191.563,97.530,-50.285,-178.838,5.997,148.728
C02525=1191.558,97.779,-50.303,-178.835,5.998,148.728
C02526=1191.553,98.028,-50.321,-178.832,5.999,148.727
C02527=1191.548,98.279,-50.340,-178.830,6.001,148.726
C02528=1191.543,98.527,-50.358,-178.827,6.001,148.726
C02529=1191.538,98.776,-50.376,-178.825,6.002,148.725
C02530=1191.533,99.026,-50.394,-178.822,6.004,148.725
C02531=1191.529,99.275,-50.413,-178.820,6.005,148.724
C02532=1191.524,99.524,-50.432,-178.817,6.006,148.724
C02533=1191.519,99.773,-50.450,-178.814,6.007,148.723
C02534=1191.514,100.023,-50.468,-178.811,6.009,148.723
C02535=1191.510,100.272,-50.487,-178.809,6.009,148.722
C02536=1191.504,100.521,-50.505,-178.806,6.011,148.722
C02537=1191.499,100.771,-50.523,-178.804,6.011,148.721
C02538=1191.495,101.020,-50.542,-178.801,6.013,148.721
C02539=1191.490,101.269,-50.561,-178.798,6.014,148.720
C02540=1191.485,101.518,-50.579,-178.795,6.015,148.720
C02541=1191.481,101.768,-50.598,-178.793,6.016,148.719
C02542=1191.475,102.017,-50.617,-178.790,6.018,148.719
C02543=1191.470,102.266,-50.635,-178.788,6.019,148.718
C02544=1191.466,102.516,-50.654,-178.785,6.020,148.718
C02545=1191.461,102.765,-50.672,-178.783,6.021,148.717
C02546=1191.456,103.014,-50.690,-178.780,6.022,148.717
C02547=1191.452,103.264,-50.709,-178.777,6.023,148.716
C02548=1191.446,103.513,-50.728,-178.775,6.024,148.716
C02549=1191.441,103.762,-50.747,-178.772,6.026,148.715
C02550=1191.437,104.011,-50.765,-178.769,6.026,148.714
C02551=1191.432,104.260,-50.784,-178.767,6.028,148.714
C02552=1191.427,104.510,-50.802,-178.765,6.029,148.714
C02553=1191.423,104.759,-50.821,-178.761,6.030,148.713
C02554=1191.417,105.008,-50.840,-178.759,6.031,148.713
C02555=1191.412,105.257,-50.859,-178.756,6.033,148.712
C02556=1191.407,105.507,-50.877,-178.754,6.034,148.712
C02557=1191.403,105.756,-50.896,-178.751,6.035,148.711
C02558=1191.398,106.005,-50.914,-178.749,6.036,148.710
C02559=1191.393,106.254,-50.934,-178.746,6.038,148.710
C02560=1191.388,106.523,-50.953,-178.743,6.039,148.709
C02561=1191.383,106.791,-50.974,-178.740,6.040,148.709
C02562=1191.377,107.060,-50.994,-178.737,6.041,148.708
C02563=1191.372,107.328,-51.014,-178.734,6.043,148.708
C02564=1191.367,107.578,-51.033,-178.732,6.044,148.707
C02565=1191.363,107.826,-51.052,-178.729,6.045,148.707
C02566=1191.358,108.076,-51.071,-178.727,6.046,148.706
C02567=1191.353,108.325,-51.090,-178.724,6.047,148.706
C02568=1191.348,108.574,-51.108,-178.721,6.048,148.705
C02569=1191.344,108.824,-51.127,-178.719,6.050,148.705
C02570=1191.338,109.072,-51.147,-178.716,6.051,148.704
C02571=1191.334,109.322,-51.165,-178.713,6.052,148.704
C02572=1191.329,109.571,-51.184,-178.711,6.053,148.703
C02573=1191.325,109.820,-51.203,-178.708,6.055,148.703
C02574=1191.319,110.070,-51.222,-178.706,6.056,148.702
C02575=1191.314,110.319,-51.241,-178.703,6.057,148.702
C02576=1191.310,110.568,-51.260,-178.700,6.059,148.701
C02577=1191.305,110.817,-51.279,-178.698,6.059,148.701
C02578=1191.300,111.067,-51.298,-178.695,6.061,148.700
C02579=1191.295,111.316,-51.317,-178.693,6.062,148.700
C02580=1191.291,111.565,-51.336,-178.689,6.063,148.699
C02581=1191.285,111.814,-51.355,-178.687,6.064,148.699
C02582=1191.281,112.064,-51.374,-178.684,6.066,148.698
C02583=1191.276,112.313,-51.393,-178.682,6.067,148.698
C02584=1191.272,112.562,-51.412,-178.679,6.068,148.697
C02585=1191.266,112.811,-51.432,-178.677,6.069,148.697
C02586=1191.261,113.061,-51.450,-178.674,6.071,148.696
C02587=1191.257,113.309,-51.469,-178.671,6.071,148.696
C02588=1191.252,113.559,-51.489,-178.669,6.073,148.695
C02589=1191.246,113.808,-51.508,-178.666,6.075,148.695
C02590=1191.242,114.057,-51.527,-178.663,6.075,148.694
C02591=1191.237,114.306,-51.546,-178.661,6.077,148.694
C02592=1191.232,114.556,-51.565,-178.658,6.078,148.693
C02593=1191.227,114.805,-51.584,-178.655,6.079,148.693
C02594=1191.223,115.054,-51.604,-178.653,6.080,148.692
C02595=1191.217,115.303,-51.623,-178.650,6.082,148.692
C02596=1191.213,115.552,-51.642,-178.647,6.083,148.691
C02597=1191.209,115.802,-51.662,-178.645,6.084,148.691
C02598=1191.203,116.051,-51.681,-178.642,6.086,148.690
C02599=1191.199,116.300,-51.700,-178.640,6.087,148.690
C02600=1191.194,116.549,-51.719,-178.637,6.088,148.689
C02601=1191.189,116.799,-51.739,-178.635,6.089,148.689
C02602=1191.184,117.047,-51.758,-178.632,6.091,148.688
C02603=1191.180,117.297,-51.777,-178.629,6.092,148.688
C02604=1191.175,117.547,-51.796,-178.627,6.093,148.687
C02605=1191.169,117.796,-51.816,-178.624,6.095,148.687
C02606=1191.165,118.045,-51.835,-178.621,6.095,148.686
C02607=1191.160,118.294,-51.854,-178.619,6.097,148.686
C02608=1191.155,118.543,-51.874,-178.616,6.098,148.686
C02609=1191.151,118.792,-51.894,-178.613,6.100,148.685
C02610=1191.146,119.041,-51.913,-178.611,6.101,148.685
C02611=1191.142,119.291,-51.932,-178.608,6.102,148.684
C02612=1191.136,119.539,-51.952,-178.605,6.104,148.684
C02613=1191.131,119.789,-51.971,-178.603,6.105,148.683
C02614=1191.127,120.039,-51.991,-178.600,6.106,148.683
C02615=1191.121,120.287,-52.010,-178.597,6.108,148.682
C02616=1191.117,120.537,-52.029,-178.595,6.109,148.682
C02617=1191.113,120.786,-52.049,-178.592,6.110,148.681
C02618=1191.107,121.035,-52.068,-178.590,6.111,148.681
C02619=1191.103,121.285,-52.088,-178.587,6.113,148.680
C02620=1191.097,121.534,-52.107,-178.584,6.114,148.680
C02621=1191.093,121.782,-52.128,-178.582,6.115,148.679
C02622=1191.089,122.032,-52.147,-178.579,6.117,148.679
C02623=1191.083,122.281,-52.166,-178.577,6.117,148.678
C02624=1191.079,122.530,-52.186,-178.574,6.119,148.678
C02625=1191.074,122.780,-52.205,-178.571,6.121,148.677
C02626=1191.069,123.028,-52.225,-178.569,6.121,148.677
C02627=1191.064,123.278,-52.245,-178.566,6.123,148.676
C02628=1191.059,123.527,-52.265,-178.564,6.124,148.676
C02629=1191.055,123.777,-52.284,-178.561,6.126,148.675
C02630=1191.050,124.025,-52.303,-178.558,6.127,148.675
C02631=1191.046,124.274,-52.323,-178.556,6.128,148.675
C02632=1191.041,124.524,-52.343,-178.553,6.130,148.674
C02633=1191.036,124.773,-52.362,-178.550,6.131,148.674
C02634=1191.031,125.022,-52.383,-178.548,6.132,148.673
C02635=1191.026,125.271,-52.402,-178.545,6.134,148.673
C02636=1191.022,125.521,-52.422,-178.542,6.135,148.672
C02637=1191.016,125.770,-52.441,-178.540,6.136,148.672
C02638=1191.012,126.019,-52.462,-178.537,6.138,148.671
C02639=1191.007,126.268,-52.481,-178.534,6.139,148.671
C02640=1191.002,126.517,-52.501,-178.532,6.141,148.670
C02641=1190.997,126.766,-52.521,-178.529,6.142,148.670
C02642=1190.993,127.015,-52.541,-178.526,6.143,148.669
C02643=1190.988,127.265,-52.560,-178.524,6.145,148.669
C02644=1190.983,127.513,-52.580,-178.522,6.146,148.668
C02645=1190.978,127.763,-52.600,-178.518,6.147,148.668
C02646=1190.974,128.012,-52.620,-178.516,6.149,148.667
C02647=1190.969,128.261,-52.640,-178.514,6.150,148.667
C02648=1190.964,128.510,-52.660,-178.510,6.151,148.666
C02649=1190.959,128.759,-52.680,-178.508,6.153,148.666
C02650=1190.954,129.009,-52.699,-178.506,6.154,148.666
C02651=1190.950,129.258,-52.720,-178.502,6.155,148.665
C02652=1190.945,129.507,-52.739,-178.500,6.157,148.665
C02653=1190.941,129.756,-52.760,-178.498,6.158,148.664
C02654=1190.935,130.005,-52.779,-178.494,6.159,148.664
C02655=1190.931,130.254,-52.799,-178.492,6.161,148.663
C02656=1190.925,130.504,-52.820,-178.490,6.162,148.663
C02657=1190.921,130.753,-52.840,-178.487,6.164,148.662
C02658=1190.916,131.002,-52.860,-178.484,6.165,148.662
C02659=1190.911,131.251,-52.880,-178.482,6.166,148.661
C02660=1190.907,131.500,-52.899,-178.479,6.168,148.661
C02661=1190.902,131.749,-52.920,-178.476,6.169,148.660
C02662=1190.897,131.999,-52.939,-178.474,6.170,148.660
C02663=1190.893,132.248,-52.960,-178.471,6.172,148.660
C02664=1190.887,132.517,-52.981,-178.468,6.173,148.659
C02665=1190.883,132.785,-53.003,-178.465,6.175,148.659
C02666=1190.877,133.054,-53.025,-178.462,6.177,148.658
C02667=1190.872,133.322,-53.047,-178.459,6.178,148.658
C02668=1190.867,133.572,-53.067,-178.457,6.179,148.657
C02669=1190.862,133.821,-53.087,-178.454,6.181,148.657
C02670=1190.858,134.069,-53.108,-178.451,6.182,148.656
C02671=1190.853,134.318,-53.127,-178.449,6.183,148.656
C02672=1190.848,134.567,-53.147,-178.446,6.185,148.655
C02673=1190.843,134.817,-53.168,-178.443,6.187,148.655
C02674=1190.838,135.066,-53.188,-178.441,6.188,148.654
C02675=1190.834,135.315,-53.208,-178.438,6.189,148.654
C02676=1190.829,135.564,-53.229,-178.436,6.191,148.654
C02677=1190.824,135.814,-53.249,-178.433,6.192,148.653
C02678=1190.820,136.063,-53.269,-178.430,6.193,148.653
C02679=1190.815,136.312,-53.290,-178.428,6.195,148.652
C02680=1190.811,136.561,-53.310,-178.425,6.197,148.652
C02681=1190.805,136.810,-53.330,-178.422,6.198,148.651
C02682=1190.800,137.059,-53.350,-178.420,6.199,148.651
C02683=1190.796,137.308,-53.371,-178.417,6.201,148.650
C02684=1190.791,137.557,-53.391,-178.415,6.202,148.650
C02685=1190.786,137.806,-53.412,-178.412,6.203,148.649
C02686=1190.781,138.056,-53.432,-178.409,6.205,148.649
C02687=1190.777,138.305,-53.452,-178.407,6.206,148.649
C02688=1190.772,138.554,-53.473,-178.404,6.208,148.648
C02689=1190.767,138.803,-53.493,-178.401,6.209,148.648
C02690=1190.763,139.052,-53.514,-178.398,6.211,148.647
C02691=1190.758,139.301,-53.535,-178.396,6.212,148.647
C02692=1190.753,139.551,-53.554,-178.394,6.214,148.646
C02693=1190.749,139.799,-53.575,-178.390,6.215,148.646
C02694=1190.743,140.049,-53.596,-178.388,6.217,148.645
C02695=1190.739,140.298,-53.616,-178.386,6.218,148.645
C02696=1190.734,140.547,-53.636,-178.383,6.220,148.645
C02697=1190.729,140.796,-53.657,-178.380,6.221,148.644
C02698=1190.725,141.045,-53.678,-178.378,6.222,148.644
C02699=1190.720,141.294,-53.699,-178.375,6.224,148.643
C02700=1190.715,141.543,-53.719,-178.372,6.226,148.643
C02701=1190.711,141.792,-53.739,-178.370,6.227,148.643
C02702=1190.706,142.041,-53.760,-178.367,6.228,148.642
C02703=1190.701,142.290,-53.781,-178.364,6.230,148.642
C02704=1190.696,142.539,-53.802,-178.362,6.231,148.641
C02705=1190.692,142.788,-53.822,-178.359,6.233,148.641
C02706=1190.686,143.038,-53.843,-178.357,6.234,148.640
C02707=1190.682,143.287,-53.863,-178.354,6.236,148.640
C02708=1190.678,143.536,-53.884,-178.351,6.237,148.639
C02709=1190.672,143.785,-53.905,-178.348,6.239,148.639
C02710=1190.668,144.034,-53.925,-178.346,6.240,148.639
C02711=1190.663,144.283,-53.946,-178.344,6.242,148.638
C02712=1190.658,144.532,-53.966,-178.340,6.243,148.638
C02713=1190.654,144.782,-53.988,-178.338,6.245,148.637
C02714=1190.649,145.031,-54.008,-178.336,6.246,148.637
C02715=1190.644,145.280,-54.029,-178.333,6.248,148.636
C02716=1190.640,145.529,-54.050,-178.330,6.250,148.636
C02717=1190.635,145.778,-54.071,-178.327,6.251,148.635
C02718=1190.630,146.027,-54.092,-178.325,6.252,148.635
C02719=1190.625,146.276,-54.113,-178.322,6.254,148.635
C02720=1190.621,146.525,-54.133,-178.320,6.255,148.634
C02721=1190.616,146.774,-54.154,-178.317,6.257,148.634
C02722=1190.611,147.023,-54.176,-178.314,6.258,148.633
C02723=1190.606,147.272,-54.196,-178.312,6.260,148.633
C02724=1190.602,147.522,-54.217,-178.309,6.261,148.633
C02725=1190.597,147.771,-54.238,-178.306,6.263,148.632
C02726=1190.592,148.020,-54.259,-178.303,6.265,148.632
C02727=1190.587,148.269,-54.280,-178.301,6.266,148.631
C02728=1190.583,148.518,-54.301,-178.298,6.267,148.631
C02729=1190.578,148.767,-54.322,-178.296,6.269,148.630
C02730=1190.573,149.016,-54.342,-178.293,6.271,148.630
C02731=1190.569,149.265,-54.364,-178.291,6.272,148.630
C02732=1190.564,149.514,-54.385,-178.288,6.274,148.629
C02733=1190.559,149.763,-54.405,-178.285,6.275,148.629
C02734=1190.554,150.012,-54.427,-178.282,6.277,148.628
C02735=1190.549,150.261,-54.448,-178.279,6.279,148.628
C02736=1190.545,150.510,-54.468,-178.277,6.279,148.627
C02737=1190.541,150.759,-54.490,-178.275,6.281,148.627
C02738=1190.535,151.009,-54.511,-178.272,6.283,148.627
C02739=1190.531,151.258,-54.532,-178.269,6.284,148.626
C02740=1190.526,151.506,-54.553,-178.266,6.286,148.626
C02741=1190.521,151.756,-54.574,-178.264,6.287,148.625
C02742=1190.517,152.004,-54.596,-178.261,6.289,148.625
C02743=1190.512,152.254,-54.617,-178.259,6.291,148.625
C02744=1190.507,152.503,-54.638,-178.256,6.293,148.624
C02745=1190.503,152.751,-54.659,-178.253,6.294,148.624
C02746=1190.498,153.001,-54.680,-178.251,6.295,148.623
C02747=1190.493,153.249,-54.702,-178.248,6.297,148.623
C02748=1190.488,153.499,-54.723,-178.245,6.298,148.622
C02749=1190.484,153.748,-54.744,-178.243,6.300,148.622
C02750=1190.479,153.997,-54.765,-178.240,6.302,148.622
C02751=1190.474,154.246,-54.787,-178.237,6.304,148.621
C02752=1190.470,154.496,-54.808,-178.235,6.304,148.621
C02753=1190.465,154.744,-54.830,-178.232,6.306,148.620
C02754=1190.460,154.993,-54.850,-178.229,6.308,148.620
C02755=1190.455,155.242,-54.872,-178.227,6.310,148.620
C02756=1190.451,155.492,-54.893,-178.224,6.311,148.619
C02757=1190.446,155.740,-54.915,-178.222,6.312,148.619
C02758=1190.441,155.990,-54.936,-178.219,6.314,148.618
C02759=1190.437,156.238,-54.957,-178.216,6.316,148.618
C02760=1190.432,156.488,-54.978,-178.213,6.317,148.617
C02761=1190.427,156.737,-55.000,-178.211,6.319,148.617
C02762=1190.422,156.985,-55.021,-178.208,6.321,148.617
C02763=1190.418,157.235,-55.043,-178.206,6.322,148.616
C02764=1190.413,157.484,-55.065,-178.203,6.324,148.616
C02765=1190.409,157.732,-55.086,-178.201,6.325,148.616
C02766=1190.404,157.982,-55.107,-178.198,6.327,148.615
C02767=1190.399,158.231,-55.129,-178.195,6.329,148.615
C02768=1190.394,158.500,-55.152,-178.192,6.330,148.614
C02769=1190.389,158.769,-55.175,-178.189,6.332,148.614
C02770=1190.384,159.038,-55.199,-178.187,6.334,148.613
C02771=1190.379,159.307,-55.222,-178.183,6.335,148.613
C02772=1190.374,159.556,-55.243,-178.181,6.337,148.613
C02773=1190.369,159.805,-55.264,-178.178,6.339,148.612
C02774=1190.365,160.054,-55.286,-178.175,6.341,148.612
C02775=1190.360,160.303,-55.308,-178.173,6.343,148.611
C02776=1190.355,160.551,-55.330,-178.171,6.344,148.611
C02777=1190.350,160.801,-55.351,-178.168,6.345,148.611
C02778=1190.346,161.050,-55.373,-178.165,6.347,148.610
C02779=1190.341,161.299,-55.394,-178.163,6.349,148.610
C02780=1190.336,161.548,-55.416,-178.159,6.350,148.609
C02781=1190.332,161.797,-55.438,-178.157,6.352,148.609
C02782=1190.327,162.046,-55.460,-178.154,6.354,148.609
C02783=1190.322,162.295,-55.481,-178.151,6.356,148.608
C02784=1190.317,162.544,-55.503,-178.149,6.357,148.608
C02785=1190.313,162.793,-55.525,-178.147,6.358,148.607
C02786=1190.308,163.042,-55.546,-178.144,6.360,148.607
C02787=1190.304,163.291,-55.569,-178.141,6.362,148.607
C02788=1190.299,163.540,-55.590,-178.139,6.364,148.606
C02789=1190.294,163.788,-55.612,-178.136,6.366,148.606
C02790=1190.290,164.038,-55.634,-178.133,6.367,148.606
C02791=1190.285,164.287,-55.655,-178.130,6.369,148.605
C02792=1190.280,164.536,-55.677,-178.128,6.370,148.605
C02793=1190.276,164.785,-55.699,-178.125,6.371,148.604
C02794=1190.271,165.034,-55.721,-178.123,6.373,148.604
C02795=1190.266,165.283,-55.742,-178.120,6.375,148.604
C02796=1190.262,165.532,-55.764,-178.117,6.377,148.603
C02797=1190.257,165.781,-55.786,-178.115,6.379,148.603
C02798=1190.252,166.030,-55.808,-178.112,6.380,148.602
C02799=1190.247,166.279,-55.830,-178.109,6.382,148.602
C02800=1190.243,166.528,-55.852,-178.107,6.384,148.602
C02801=1190.238,166.777,-55.874,-178.104,6.386,148.601
C02802=1190.233,167.026,-55.896,-178.102,6.387,148.601
C02803=1190.229,167.275,-55.918,-178.099,6.388,148.601
C02804=1190.224,167.524,-55.940,-178.096,6.390,148.600
C02805=1190.220,167.773,-55.963,-178.094,6.392,148.600
C02806=1190.215,168.022,-55.985,-178.091,6.394,148.599
C02807=1190.210,168.271,-56.007,-178.088,6.395,148.599
C02808=1190.206,168.520,-56.028,-178.085,6.397,148.598
C02809=1190.201,168.769,-56.050,-178.083,6.399,148.598
C02810=1190.196,169.018,-56.072,-178.080,6.401,148.598
C02811=1190.191,169.267,-56.095,-178.077,6.402,148.597
C02812=1190.187,169.516,-56.116,-178.075,6.404,148.597
C02813=1190.183,169.765,-56.139,-178.072,6.406,148.597
C02814=1190.178,170.013,-56.161,-178.070,6.407,148.596
C02815=1190.173,170.263,-56.183,-178.067,6.409,148.596
C02816=1190.168,170.512,-56.205,-178.064,6.411,148.596
C02817=1190.164,170.761,-56.227,-178.062,6.412,148.595
C02818=1190.159,171.009,-56.249,-178.059,6.414,148.595
C02819=1190.154,171.259,-56.272,-178.056,6.416,148.594
C02820=1190.150,171.508,-56.294,-178.054,6.418,148.594
C02821=1190.145,171.757,-56.316,-178.051,6.419,148.594
C02822=1190.141,172.006,-56.338,-178.048,6.421,148.593
C02823=1190.135,172.254,-56.361,-178.046,6.423,148.593
C02824=1190.131,172.504,-56.383,-178.043,6.425,148.593
C02825=1190.126,172.752,-56.405,-178.040,6.427,148.592
C02826=1190.121,173.001,-56.428,-178.038,6.428,148.592
C02827=1190.117,173.251,-56.450,-178.035,6.430,148.592
C02828=1190.112,173.499,-56.472,-178.032,6.432,148.591
C02829=1190.108,173.748,-56.495,-178.030,6.434,148.591
C02830=1190.103,173.997,-56.517,-178.028,6.435,148.590
C02831=1190.098,174.246,-56.539,-178.025,6.436,148.590
C02832=1190.094,174.495,-56.562,-178.022,6.438,148.590
C02833=1190.089,174.744,-56.584,-178.020,6.440,148.589
C02834=1190.085,174.993,-56.606,-178.017,6.442,148.589
C02835=1190.079,175.242,-56.629,-178.014,6.444,148.589
C02836=1190.075,175.491,-56.651,-178.012,6.445,148.588
C02837=1190.070,175.740,-56.674,-178.009,6.447,148.588
C02838=1190.066,175.989,-56.696,-178.006,6.449,148.588
C02839=1190.062,176.237,-56.719,-178.004,6.451,148.587
C02840=1190.057,176.487,-56.742,-178.001,6.453,148.587
C02841=1190.052,176.736,-56.763,-177.998,6.454,148.586
C02842=1190.047,176.985,-56.787,-177.996,6.456,148.586
C02843=1190.043,177.234,-56.809,-177.993,6.458,148.586
C02844=1190.037,177.482,-56.832,-177.990,6.460,148.585
C02845=1190.033,177.732,-56.854,-177.988,6.462,148.585
C02846=1190.029,177.980,-56.876,-177.985,6.463,148.585
C02847=1190.024,178.229,-56.899,-177.982,6.465,148.584
C02848=1190.020,178.478,-56.921,-177.980,6.467,148.584
C02849=1190.015,178.727,-56.945,-177.977,6.469,148.584
C02850=1190.010,178.976,-56.967,-177.974,6.470,148.583
C02851=1190.005,179.225,-56.990,-177.972,6.472,148.583
C02852=1190.001,179.474,-57.012,-177.969,6.474,148.582
C02853=1189.996,179.723,-57.035,-177.966,6.476,148.582
C02854=1189.992,179.971,-57.058,-177.963,6.478,148.582
C02855=1189.987,180.221,-57.080,-177.961,6.479,148.581
C02856=1189.983,180.469,-57.103,-177.958,6.481,148.581
C02857=1189.977,180.718,-57.125,-177.955,6.483,148.581
C02858=1189.973,180.967,-57.149,-177.953,6.485,148.580
C02859=1189.969,181.216,-57.171,-177.950,6.487,148.580
C02860=1189.964,181.466,-57.194,-177.947,6.488,148.580
C02861=1189.959,181.714,-57.217,-177.945,6.490,148.579
C02862=1189.954,181.963,-57.240,-177.942,6.492,148.579
C02863=1189.950,182.212,-57.263,-177.939,6.494,148.579
C02864=1189.945,182.461,-57.285,-177.937,6.496,148.578
C02865=1189.941,182.710,-57.309,-177.934,6.497,148.578
C02866=1189.936,182.958,-57.331,-177.931,6.499,148.577
C02867=1189.931,183.208,-57.354,-177.929,6.501,148.577
C02868=1189.927,183.457,-57.376,-177.927,6.503,148.577
C02869=1189.922,183.706,-57.400,-177.924,6.505,148.577
C02870=1189.917,183.954,-57.423,-177.921,6.507,148.576
C02871=1189.913,184.203,-57.446,-177.919,6.508,148.576
C02872=1189.908,184.473,-57.471,-177.916,6.510,148.576
C02873=1189.903,184.742,-57.495,-177.913,6.513,148.575
C02874=1189.898,185.012,-57.520,-177.910,6.514,148.575
C02875=1189.893,185.282,-57.545,-177.907,6.516,148.574
C02876=1189.889,185.530,-57.568,-177.904,6.518,148.574
C02877=1189.884,185.779,-57.591,-177.902,6.520,148.574
C02878=1189.879,186.028,-57.615,-177.899,6.522,148.573
C02879=1189.874,186.278,-57.637,-177.897,6.524,148.573
C02880=1189.870,186.526,-57.660,-177.894,6.525,148.573
C02881=1189.865,186.775,-57.683,-177.891,6.527,148.572
C02882=1189.860,187.024,-57.706,-177.889,6.529,148.572
C02883=1189.856,187.273,-57.729,-177.886,6.531,148.572
C02884=1189.852,187.522,-57.752,-177.883,6.533,148.571
C02885=1189.847,187.771,-57.776,-177.881,6.534,148.571
C02886=1189.842,188.020,-57.799,-177.877,6.537,148.571
C02887=1189.838,188.268,-57.822,-177.875,6.539,148.570
C02888=1189.833,188.517,-57.845,-177.872,6.541,148.570
C02889=1189.828,188.766,-57.868,-177.870,6.543,148.570
C02890=1189.824,189.015,-57.892,-177.867,6.545,148.569
C02891=1189.819,189.264,-57.915,-177.865,6.546,148.569
C02892=1189.815,189.513,-57.938,-177.862,6.548,148.569
C02893=1189.810,189.762,-57.961,-177.859,6.550,148.568
C02894=1189.805,190.011,-57.985,-177.857,6.552,148.568
C02895=1189.801,190.260,-58.008,-177.854,6.554,148.568
C02896=1189.795,190.508,-58.031,-177.851,6.555,148.567
C02897=1189.791,190.757,-58.054,-177.849,6.557,148.567
C02898=1189.787,191.006,-58.077,-177.846,6.559,148.567
C02899=1189.782,191.254,-58.101,-177.844,6.561,148.567
C02900=1189.778,191.503,-58.124,-177.841,6.563,148.566
C02901=1189.773,191.752,-58.148,-177.838,6.565,148.566
C02902=1189.768,192.001,-58.171,-177.835,6.567,148.565
C02903=1189.764,192.250,-58.194,-177.833,6.569,148.565
C02904=1189.759,192.499,-58.218,-177.830,6.571,148.565
C02905=1189.755,192.748,-58.242,-177.827,6.573,148.564
C02906=1189.750,192.997,-58.265,-177.825,6.575,148.564
C02907=1189.745,193.246,-58.289,-177.822,6.576,148.564
C02908=1189.741,193.495,-58.311,-177.820,6.578,148.564
C02909=1189.736,193.744,-58.335,-177.817,6.580,148.563
C02910=1189.732,193.992,-58.359,-177.814,6.582,148.563
C02911=1189.727,194.241,-58.382,-177.812,6.584,148.563
C02912=1189.723,194.490,-58.406,-177.809,6.586,148.562
C02913=1189.718,194.739,-58.429,-177.806,6.587,148.562
C02914=1189.714,194.988,-58.453,-177.803,6.590,148.562
C02915=1189.709,195.237,-58.476,-177.801,6.592,148.561
C02916=1189.704,195.486,-58.500,-177.798,6.594,148.561
C02917=1189.700,195.734,-58.524,-177.796,6.596,148.561
C02918=1189.695,195.983,-58.547,-177.793,6.598,148.560
C02919=1189.690,196.232,-58.570,-177.790,6.599,148.560
C02920=1189.686,196.481,-58.595,-177.788,6.601,148.560
C02921=1189.681,196.730,-58.618,-177.785,6.603,148.559
C02922=1189.677,196.979,-58.641,-177.783,6.605,148.559
C02923=1189.672,197.227,-58.665,-177.780,6.608,148.559
C02924=1189.668,197.476,-58.689,-177.777,6.610,148.559
C02925=1189.663,197.725,-58.713,-177.774,6.611,148.558
C02926=1189.658,197.974,-58.736,-177.772,6.613,148.558
C02927=1189.654,198.223,-58.760,-177.769,6.615,148.557
C02928=1189.649,198.471,-58.784,-177.766,6.617,148.557
C02929=1189.644,198.720,-58.808,-177.764,6.619,148.557
C02930=1189.639,198.969,-58.832,-177.761,6.621,148.557
C02931=1189.635,199.218,-58.855,-177.759,6.623,148.556
C02932=1189.630,199.466,-58.879,-177.756,6.625,148.556
C02933=1189.626,199.716,-58.903,-177.753,6.627,148.556
C02934=1189.622,199.964,-58.927,-177.750,6.629,148.555
C02935=1189.617,200.213,-58.950,-177.748,6.631,148.555
C02936=1189.613,200.462,-58.974,-177.745,6.633,148.555
C02937=1189.607,200.711,-58.998,-177.743,6.635,148.554
C02938=1189.603,200.960,-59.022,-177.740,6.636,148.554
C02939=1189.598,201.209,-59.046,-177.737,6.639,148.554
C02940=1189.594,201.457,-59.070,-177.735,6.641,148.554
C02941=1189.589,201.705,-59.094,-177.732,6.643,148.553
C02942=1189.585,201.955,-59.118,-177.729,6.645,148.553
C02943=1189.580,202.204,-59.142,-177.727,6.647,148.553
C02944=1189.576,202.453,-59.166,-177.724,6.648,148.552
C02945=1189.571,202.701,-59.190,-177.721,6.650,148.552
C02946=1189.567,202.950,-59.214,-177.719,6.653,148.552
C02947=1189.562,203.199,-59.237,-177.716,6.655,148.552
C02948=1189.557,203.447,-59.262,-177.713,6.657,148.551
C02949=1189.553,203.697,-59.286,-177.711,6.659,148.551
C02950=1189.548,203.946,-59.310,-177.708,6.660,148.551
C02951=1189.544,204.194,-59.334,-177.706,6.662,148.550
C02952=1189.539,204.443,-59.358,-177.703,6.665,148.550
C02953=1189.535,204.691,-59.382,-177.700,6.667,148.550
C02954=1189.530,204.941,-59.406,-177.697,6.669,148.549
C02955=1189.526,205.189,-59.430,-177.695,6.671,148.549
C02956=1189.521,205.438,-59.455,-177.692,6.673,148.549
C02957=1189.517,205.686,-59.479,-177.690,6.674,148.549
C02958=1189.512,205.935,-59.502,-177.687,6.677,148.548
C02959=1189.507,206.185,-59.527,-177.684,6.679,148.548
C02960=1189.503,206.433,-59.551,-177.682,6.681,148.548
C02961=1189.498,206.682,-59.575,-177.679,6.683,148.547
C02962=1189.493,206.930,-59.600,-177.676,6.685,148.547
C02963=1189.489,207.179,-59.623,-177.674,6.686,148.547
C02964=1189.485,207.429,-59.648,-177.671,6.689,148.546
C02965=1189.480,207.677,-59.673,-177.668,6.691,148.546
C02966=1189.475,207.926,-59.697,-177.666,6.693,148.546
C02967=1189.470,208.174,-59.721,-177.663,6.695,148.546
C02968=1189.466,208.424,-59.746,-177.660,6.697,148.545
C02969=1189.462,208.672,-59.770,-177.658,6.700,148.545
C02970=1189.457,208.921,-59.795,-177.655,6.701,148.545
C02971=1189.452,209.169,-59.819,-177.652,6.703,148.545
C02972=1189.448,209.419,-59.844,-177.650,6.705,148.544
C02973=1189.444,209.667,-59.868,-177.648,6.707,148.544
C02974=1189.439,209.916,-59.891,-177.644,6.710,148.544
C02975=1189.434,210.165,-59.916,-177.642,6.712,148.543
C02976=1189.429,210.436,-59.943,-177.639,6.713,148.543
C02977=1189.424,210.706,-59.970,-177.636,6.716,148.543
C02978=1189.420,210.976,-59.996,-177.633,6.718,148.542
C02979=1189.415,211.246,-60.023,-177.630,6.721,148.542
C02980=1189.410,211.495,-60.047,-177.628,6.723,148.542
C02981=1189.406,211.744,-60.071,-177.625,6.724,148.542
C02982=1189.401,211.993,-60.096,-177.622,6.726,148.541
C02983=1189.397,212.241,-60.121,-177.620,6.728,148.541
C02984=1189.391,212.490,-60.145,-177.617,6.731,148.541
C02985=1189.388,212.739,-60.170,-177.614,6.733,148.541
C02986=1189.383,212.988,-60.194,-177.612,6.735,148.540
C02987=1189.378,213.236,-60.218,-177.610,6.737,148.540
C02988=1189.374,213.485,-60.244,-177.606,6.739,148.540
C02989=1189.370,213.734,-60.268,-177.604,6.741,148.540
C02990=1189.364,213.982,-60.293,-177.601,6.743,148.539
C02991=1189.360,214.232,-60.318,-177.599,6.745,148.539
C02992=1189.355,214.480,-60.342,-177.596,6.748,148.539
C02993=1189.350,214.729,-60.367,-177.593,6.750,148.538
C02994=1189.347,214.977,-60.392,-177.590,6.752,148.538
C02995=1189.342,215.226,-60.417,-177.588,6.754,148.538
C02996=1189.338,215.475,-60.441,-177.586,6.755,148.538
C02997=1189.333,215.724,-60.466,-177.582,6.758,148.537
C02998=1189.328,215.972,-60.491,-177.580,6.760,148.537
C02999=1189.324,216.221,-60.515,-177.577,6.762,148.537
C03000=1189.319,216.470,-60.540,-177.575,6.764,148.537
C03001=1189.315,216.719,-60.565,-177.572,6.767,148.536
C03002=1189.310,216.967,-60.590,-177.569,6.769,148.536
C03003=1189.306,217.217,-60.615,-177.567,6.770,148.536
C03004=1189.301,217.465,-60.640,-177.564,6.772,148.535
C03005=1189.297,217.713,-60.664,-177.561,6.775,148.535
C03006=1189.292,217.963,-60.689,-177.559,6.777,148.535
C03007=1189.287,218.211,-60.714,-177.556,6.779,148.535
C03008=1189.284,218.460,-60.739,-177.554,6.781,148.535
C03009=1189.278,218.708,-60.764,-177.551,6.784,148.534
C03010=1189.274,218.958,-60.789,-177.548,6.785,148.534
C03011=1189.270,219.206,-60.814,-177.546,6.788,148.534
C03012=1189.265,219.455,-60.839,-177.543,6.789,148.534
C03013=1189.260,219.703,-60.864,-177.540,6.792,148.533
C03014=1189.256,219.953,-60.889,-177.538,6.794,148.533
C03015=1189.252,220.200,-60.914,-177.535,6.796,148.533
C03016=1189.247,220.450,-60.939,-177.533,6.798,148.532
C03017=1189.242,220.698,-60.964,-177.530,6.801,148.532
C03018=1189.238,220.947,-60.990,-177.527,6.803,148.532
C03019=1189.234,221.195,-61.014,-177.524,6.804,148.532
C03020=1189.229,221.445,-61.039,-177.522,6.807,148.532
C03021=1189.224,221.693,-61.065,-177.519,6.809,148.531
C03022=1189.220,221.942,-61.090,-177.516,6.811,148.531
C03023=1189.215,222.190,-61.115,-177.514,6.813,148.531
C03024=1189.211,222.439,-61.140,-177.511,6.816,148.531
C03025=1189.207,222.687,-61.165,-177.508,6.818,148.530
C03026=1189.202,222.937,-61.190,-177.506,6.820,148.530
C03027=1189.197,223.185,-61.215,-177.504,6.822,148.530
C03028=1189.193,223.434,-61.241,-177.500,6.824,148.529
C03029=1189.188,223.682,-61.266,-177.498,6.826,148.529
C03030=1189.184,223.931,-61.291,-177.496,6.828,148.529
C03031=1189.179,224.180,-61.316,-177.492,6.831,148.529
C03032=1189.175,224.429,-61.341,-177.490,6.833,148.529
C03033=1189.171,224.677,-61.367,-177.488,6.835,148.528
C03034=1189.166,224.926,-61.392,-177.485,6.837,148.528
C03035=1189.161,225.175,-61.418,-177.482,6.840,148.528
C03036=1189.157,225.423,-61.443,-177.479,6.841,148.528
C03037=1189.152,225.672,-61.468,-177.477,6.844,148.527
C03038=1189.147,225.920,-61.493,-177.474,6.846,148.527
C03039=1189.143,226.169,-61.519,-177.471,6.848,148.527
C03040=1189.139,226.418,-61.545,-177.469,6.850,148.527
C03041=1189.134,226.666,-61.569,-177.466,6.853,148.526
C03042=1189.130,226.915,-61.595,-177.464,6.855,148.526
C03043=1189.126,227.164,-61.620,-177.461,6.857,148.526
C03044=1189.121,227.412,-61.646,-177.459,6.859,148.526
C03045=1189.117,227.661,-61.672,-177.456,6.862,148.526
C03046=1189.112,227.910,-61.696,-177.453,6.863,148.525
C03047=1189.107,228.159,-61.722,-177.451,6.866,148.525
C03048=1189.103,228.407,-61.748,-177.448,6.868,148.525
C03049=1189.098,228.655,-61.773,-177.445,6.870,148.525
C03050=1189.094,228.904,-61.799,-177.443,6.872,148.524
C03051=1189.090,229.153,-61.825,-177.440,6.875,148.524
C03052=1189.085,229.402,-61.849,-177.438,6.877,148.524
C03053=1189.080,229.651,-61.876,-177.435,6.879,148.524
C03054=1189.076,229.900,-61.901,-177.432,6.882,148.523
C03055=1189.071,230.148,-61.927,-177.430,6.884,148.523
C03056=1189.067,230.397,-61.953,-177.427,6.885,148.523
C03057=1189.062,230.645,-61.978,-177.424,6.888,148.523
C03058=1189.058,230.894,-62.004,-177.422,6.890,148.523
C03059=1189.053,231.142,-62.029,-177.419,6.892,148.522
C03060=1189.049,231.391,-62.055,-177.416,6.895,148.522
C03061=1189.044,231.639,-62.081,-177.414,6.897,148.522
C03062=1189.040,231.888,-62.106,-177.411,6.899,148.522
C03063=1189.036,232.137,-62.132,-177.408,6.902,148.521
C03064=1189.031,232.386,-62.158,-177.406,6.904,148.521
C03065=1189.026,232.634,-62.184,-177.403,6.906,148.521
C03066=1189.022,232.883,-62.210,-177.401,6.909,148.521
C03067=1189.018,233.132,-62.235,-177.398,6.910,148.521
C03068=1189.013,233.380,-62.261,-177.396,6.913,148.521
C03069=1189.009,233.629,-62.286,-177.393,6.915,148.520
C03070=1189.004,233.877,-62.312,-177.390,6.917,148.520
C03071=1189.000,234.126,-62.339,-177.388,6.919,148.520
C03072=1188.995,234.375,-62.365,-177.385,6.922,148.520
C03073=1188.991,234.623,-62.390,-177.382,6.924,148.519
C03074=1188.986,234.872,-62.416,-177.380,6.926,148.519
C03075=1188.982,235.120,-62.442,-177.377,6.929,148.519
C03076=1188.977,235.370,-62.468,-177.374,6.931,148.519
C03077=1188.972,235.618,-62.494,-177.372,6.934,148.519
C03078=1188.968,235.866,-62.520,-177.369,6.935,148.518
C03079=1188.964,236.115,-62.546,-177.367,6.938,148.518
C03080=1188.959,236.387,-62.574,-177.364,6.940,148.518
C03081=1188.954,236.657,-62.603,-177.360,6.943,148.518
C03082=1188.949,236.929,-62.631,-177.358,6.945,148.518
C03083=1188.945,237.201,-62.660,-177.355,6.948,148.517
C03084=1188.940,237.450,-62.686,-177.353,6.950,148.517
C03085=1188.936,237.698,-62.712,-177.350,6.953,148.517
C03086=1188.931,237.947,-62.737,-177.348,6.955,148.517
C03087=1188.926,238.195,-62.764,-177.345,6.957,148.516
C03088=1188.922,238.444,-62.790,-177.342,6.960,148.516
C03089=1188.918,238.693,-62.816,-177.339,6.961,148.516
C03090=1188.913,238.941,-62.843,-177.337,6.964,148.516
C03091=1188.909,239.190,-62.868,-177.334,6.966,148.516
C03092=1188.904,239.438,-62.894,-177.332,6.968,148.516
C03093=1188.899,239.687,-62.921,-177.329,6.971,148.515
C03094=1188.895,239.935,-62.947,-177.327,6.973,148.515
C03095=1188.891,240.184,-62.973,-177.323,6.976,148.515
C03096=1188.886,240.433,-63.000,-177.321,6.978,148.515
C03097=1188.882,240.682,-63.025,-177.319,6.980,148.514
C03098=1188.877,240.930,-63.052,-177.316,6.983,148.514
C03099=1188.873,241.179,-63.078,-177.313,6.985,148.514
C03100=1188.869,241.426,-63.104,-177.310,6.988,148.514
C03101=1188.864,241.675,-63.131,-177.308,6.989,148.514
C03102=1188.860,241.924,-63.157,-177.306,6.992,148.514
C03103=1188.855,242.173,-63.183,-177.302,6.994,148.513
C03104=1188.851,242.421,-63.210,-177.300,6.996,148.513
C03105=1188.846,242.670,-63.236,-177.297,6.999,148.513
C03106=1188.842,242.918,-63.263,-177.295,7.001,148.513
C03107=1188.837,243.167,-63.289,-177.293,7.003,148.513
C03108=1188.833,243.415,-63.315,-177.290,7.006,148.512
C03109=1188.828,243.664,-63.342,-177.287,7.008,148.512
C03110=1188.824,243.913,-63.368,-177.284,7.011,148.512
C03111=1188.819,244.161,-63.395,-177.282,7.013,148.512
C03112=1188.815,244.410,-63.421,-177.279,7.015,148.512
C03113=1188.811,244.659,-63.448,-177.277,7.018,148.512
C03114=1188.807,244.907,-63.475,-177.274,7.020,148.511
C03115=1188.802,245.156,-63.501,-177.271,7.023,148.511
C03116=1188.797,245.403,-63.527,-177.269,7.025,148.511
C03117=1188.793,245.652,-63.554,-177.266,7.027,148.511
C03118=1188.788,245.901,-63.580,-177.264,7.030,148.511
C03119=1188.784,246.149,-63.607,-177.261,7.031,148.510
C03120=1188.780,246.397,-63.633,-177.258,7.034,148.510
C03121=1188.775,246.646,-63.660,-177.256,7.036,148.510
C03122=1188.770,246.895,-63.687,-177.253,7.039,148.510
C03123=1188.766,247.143,-63.713,-177.251,7.041,148.510
C03124=1188.762,247.392,-63.740,-177.248,7.044,148.510
C03125=1188.757,247.640,-63.766,-177.245,7.046,148.510
C03126=1188.753,247.889,-63.793,-177.242,7.049,148.509
C03127=1188.748,248.137,-63.820,-177.240,7.051,148.509
C03128=1188.745,248.386,-63.847,-177.238,7.053,148.509
C03129=1188.740,248.635,-63.873,-177.235,7.056,148.509
C03130=1188.735,248.884,-63.900,-177.233,7.058,148.509
C03131=1188.731,249.132,-63.927,-177.230,7.061,148.509
C03132=1188.726,249.381,-63.954,-177.227,7.063,148.508
C03133=1188.722,249.629,-63.981,-177.224,7.066,148.508
C03134=1188.718,249.877,-64.007,-177.222,7.068,148.508
C03135=1188.713,250.126,-64.035,-177.219,7.071,148.508
C03136=1188.708,250.375,-64.061,-177.217,7.073,148.508
C03137=1188.704,250.623,-64.087,-177.214,7.075,148.508
C03138=1188.700,250.872,-64.114,-177.212,7.077,148.507
C03139=1188.695,251.120,-64.141,-177.208,7.080,148.507
C03140=1188.690,251.369,-64.169,-177.206,7.082,148.507
C03141=1188.686,251.617,-64.195,-177.204,7.084,148.507
C03142=1188.682,251.865,-64.222,-177.201,7.087,148.507
C03143=1188.678,252.114,-64.249,-177.199,7.089,148.507
C03144=1188.673,252.363,-64.277,-177.196,7.092,148.507
C03145=1188.669,252.611,-64.303,-177.193,7.094,148.506
C03146=1188.665,252.860,-64.330,-177.191,7.097,148.506
C03147=1188.660,253.108,-64.357,-177.188,7.099,148.506
C03148=1188.655,253.357,-64.384,-177.185,7.102,148.506
C03149=1188.651,253.605,-64.411,-177.183,7.104,148.506
C03150=1188.647,253.853,-64.438,-177.180,7.107,148.506
C03151=1188.643,254.103,-64.465,-177.178,7.109,148.505
C03152=1188.638,254.351,-64.492,-177.175,7.112,148.505
C03153=1188.634,254.599,-64.520,-177.173,7.114,148.505
C03154=1188.629,254.847,-64.547,-177.170,7.117,148.505
C03155=1188.624,255.096,-64.574,-177.167,7.119,148.505
C03156=1188.620,255.344,-64.601,-177.165,7.122,148.505
C03157=1188.616,255.593,-64.628,-177.162,7.124,148.504
C03158=1188.612,255.842,-64.655,-177.159,7.127,148.504
C03159=1188.607,256.090,-64.682,-177.157,7.129,148.504
C03160=1188.603,256.338,-64.710,-177.154,7.131,148.504
C03161=1188.598,256.587,-64.737,-177.152,7.134,148.504
C03162=1188.593,256.835,-64.764,-177.149,7.137,148.504
C03163=1188.589,257.084,-64.791,-177.147,7.138,148.504
C03164=1188.585,257.333,-64.819,-177.144,7.141,148.504
C03165=1188.580,257.581,-64.846,-177.142,7.144,148.503
C03166=1188.576,257.829,-64.873,-177.138,7.146,148.503
C03167=1188.572,258.078,-64.901,-177.136,7.148,148.503
C03168=1188.568,258.326,-64.928,-177.134,7.151,148.503
C03169=1188.563,258.574,-64.955,-177.131,7.154,148.503
C03170=1188.559,258.823,-64.982,-177.128,7.156,148.503
C03171=1188.554,259.071,-65.009,-177.125,7.159,148.503
C03172=1188.550,259.320,-65.037,-177.123,7.161,148.503
C03173=1188.546,259.568,-65.064,-177.120,7.164,148.502
C03174=1188.541,259.816,-65.092,-177.118,7.166,148.502
C03175=1188.537,260.065,-65.119,-177.115,7.169,148.502
C03176=1188.532,260.314,-65.147,-177.113,7.171,148.502
C03177=1188.528,260.562,-65.174,-177.110,7.174,148.502
C03178=1188.523,260.811,-65.202,-177.108,7.176,148.502
C03179=1188.519,261.059,-65.230,-177.105,7.179,148.502
C03180=1188.514,261.308,-65.257,-177.102,7.181,148.501
C03181=1188.510,261.556,-65.284,-177.100,7.184,148.501
C03182=1188.505,261.804,-65.312,-177.097,7.186,148.501
C03183=1188.501,262.053,-65.340,-177.095,7.189,148.501
C03184=1188.496,262.326,-65.370,-177.092,7.192,148.501
C03185=1188.492,262.599,-65.400,-177.089,7.195,148.501
C03186=1188.487,262.872,-65.430,-177.086,7.198,148.501
C03187=1188.482,263.145,-65.461,-177.083,7.200,148.501
C03188=1188.478,263.393,-65.489,-177.081,7.203,148.500
C03189=1188.473,263.641,-65.516,-177.078,7.206,148.500
C03190=1188.469,263.890,-65.544,-177.075,7.207,148.500
C03191=1188.465,264.138,-65.571,-177.073,7.210,148.500
C03192=1188.460,264.387,-65.599,-177.070,7.213,148.500
C03193=1188.456,264.635,-65.627,-177.068,7.216,148.500
C03194=1188.451,264.884,-65.655,-177.065,7.217,148.500
C03195=1188.447,265.132,-65.682,-177.062,7.220,148.500
C03196=1188.443,265.381,-65.710,-177.060,7.223,148.500
C03197=1188.438,265.629,-65.737,-177.058,7.226,148.499
C03198=1188.433,265.877,-65.766,-177.055,7.229,148.499
C03199=1188.429,266.126,-65.793,-177.052,7.230,148.499
C03200=1188.425,266.374,-65.821,-177.049,7.233,148.499
C03201=1188.421,266.622,-65.849,-177.047,7.236,148.499
C03202=1188.416,266.871,-65.878,-177.045,7.239,148.499
C03203=1188.412,267.119,-65.905,-177.041,7.241,148.499
C03204=1188.408,267.368,-65.933,-177.039,7.243,148.499
C03205=1188.403,267.616,-65.961,-177.037,7.246,148.499
C03206=1188.399,267.864,-65.989,-177.034,7.249,148.498
C03207=1188.394,268.113,-66.016,-177.032,7.252,148.498
C03208=1188.390,268.361,-66.044,-177.028,7.254,148.498
C03209=1188.385,268.610,-66.073,-177.026,7.256,148.498
C03210=1188.381,268.858,-66.101,-177.024,7.259,148.498
C03211=1188.377,269.107,-66.128,-177.021,7.262,148.498
C03212=1188.373,269.355,-66.156,-177.019,7.265,148.498
C03213=1188.368,269.604,-66.185,-177.015,7.267,148.498
C03214=1188.364,269.851,-66.212,-177.013,7.269,148.498
C03215=1188.359,270.100,-66.241,-177.011,7.272,148.497
C03216=1188.355,270.348,-66.269,-177.008,7.275,148.497
C03217=1188.351,270.596,-66.297,-177.006,7.278,148.497
C03218=1188.346,270.845,-66.325,-177.003,7.281,148.497
C03219=1188.342,271.093,-66.353,-177.000,7.282,148.497
C03220=1188.338,271.342,-66.381,-176.998,7.285,148.497
C03221=1188.333,271.590,-66.409,-176.995,7.288,148.497
C03222=1188.329,271.839,-66.437,-176.993,7.291,148.497
C03223=1188.324,272.087,-66.465,-176.990,7.294,148.497
C03224=1188.320,272.336,-66.494,-176.988,7.296,148.497
C03225=1188.316,272.583,-66.521,-176.985,7.298,148.496
C03226=1188.311,272.832,-66.550,-176.982,7.301,148.496
C03227=1188.307,273.080,-66.578,-176.980,7.303,148.496
C03228=1188.302,273.329,-66.607,-176.977,7.306,148.496
C03229=1188.298,273.577,-66.634,-176.975,7.309,148.496
C03230=1188.294,273.826,-66.663,-176.972,7.312,148.496
C03231=1188.290,274.074,-66.692,-176.969,7.314,148.496
C03232=1188.285,274.322,-66.720,-176.967,7.316,148.496
C03233=1188.281,274.571,-66.749,-176.964,7.319,148.496
C03234=1188.276,274.819,-66.777,-176.961,7.322,148.496
C03235=1188.272,275.067,-66.805,-176.959,7.325,148.496
C03236=1188.267,275.316,-66.833,-176.957,7.328,148.496
C03237=1188.264,275.564,-66.862,-176.954,7.330,148.496
C03238=1188.259,275.812,-66.890,-176.952,7.333,148.496
C03239=1188.255,276.060,-66.919,-176.949,7.335,148.495
C03240=1188.251,276.309,-66.948,-176.946,7.338,148.495
C03241=1188.246,276.557,-66.975,-176.944,7.341,148.495
C03242=1188.242,276.806,-67.004,-176.941,7.344,148.495
C03243=1188.237,277.054,-67.032,-176.939,7.346,148.495
C03244=1188.233,277.302,-67.061,-176.936,7.349,148.495
C03245=1188.229,277.551,-67.090,-176.933,7.352,148.495
C03246=1188.224,277.799,-67.118,-176.931,7.354,148.495
C03247=1188.220,278.048,-67.147,-176.928,7.357,148.495
C03248=1188.216,278.296,-67.175,-176.925,7.360,148.495
C03249=1188.211,278.544,-67.204,-176.923,7.362,148.495
C03250=1188.207,278.793,-67.233,-176.920,7.365,148.494
C03251=1188.203,279.040,-67.261,-176.918,7.368,148.494
C03252=1188.198,279.289,-67.290,-176.915,7.370,148.494
C03253=1188.195,279.537,-67.318,-176.913,7.373,148.494
C03254=1188.190,279.785,-67.347,-176.910,7.376,148.494
C03255=1188.185,280.034,-67.376,-176.908,7.378,148.494
C03256=1188.182,280.282,-67.405,-176.905,7.381,148.494
C03257=1188.177,280.530,-67.433,-176.902,7.384,148.494
C03258=1188.172,280.779,-67.462,-176.900,7.386,148.494
C03259=1188.169,281.027,-67.491,-176.897,7.389,148.494
C03260=1188.164,281.275,-67.519,-176.894,7.392,148.494
C03261=1188.160,281.523,-67.548,-176.892,7.394,148.494
C03262=1188.155,281.772,-67.577,-176.890,7.397,148.494
C03263=1188.152,282.020,-67.606,-176.887,7.400,148.494
C03264=1188.147,282.268,-67.634,-176.885,7.402,148.494
C03265=1188.142,282.517,-67.664,-176.882,7.405,148.494
C03266=1188.138,282.766,-67.693,-176.879,7.408,148.493
C03267=1188.134,283.013,-67.721,-176.877,7.410,148.493
C03268=1188.129,283.262,-67.750,-176.874,7.413,148.493
C03269=1188.125,283.510,-67.779,-176.872,7.416,148.493
C03270=1188.121,283.759,-67.808,-176.869,7.419,148.493
C03271=1188.116,284.006,-67.837,-176.867,7.422,148.493
C03272=1188.112,284.255,-67.865,-176.864,7.425,148.493
C03273=1188.108,284.503,-67.895,-176.861,7.428,148.493
C03274=1188.103,284.751,-67.924,-176.859,7.430,148.493
C03275=1188.099,285.000,-67.952,-176.856,7.433,148.493
C03276=1188.095,285.248,-67.982,-176.853,7.435,148.493
C03277=1188.090,285.496,-68.011,-176.851,7.438,148.493
C03278=1188.087,285.745,-68.040,-176.848,7.441,148.493
C03279=1188.082,285.992,-68.069,-176.846,7.444,148.493
C03280=1188.078,286.241,-68.098,-176.844,7.446,148.493
C03281=1188.073,286.490,-68.127,-176.841,7.449,148.493
C03282=1188.069,286.738,-68.156,-176.838,7.452,148.493
C03283=1188.064,286.985,-68.185,-176.835,7.455,148.493
C03284=1188.060,287.234,-68.214,-176.833,7.457,148.492
C03285=1188.056,287.483,-68.244,-176.831,7.460,148.492
C03286=1188.051,287.731,-68.273,-176.828,7.463,148.492
C03287=1188.047,287.979,-68.302,-176.826,7.465,148.492
C03288=1188.042,288.253,-68.334,-176.822,7.469,148.492
C03289=1188.038,288.528,-68.366,-176.820,7.472,148.492
C03290=1188.033,288.803,-68.399,-176.817,7.475,148.492
C03291=1188.028,289.077,-68.431,-176.814,7.478,148.492
C03292=1188.024,289.325,-68.460,-176.812,7.481,148.492
C03293=1188.020,289.573,-68.490,-176.809,7.483,148.492
C03294=1188.016,289.822,-68.519,-176.807,7.486,148.492
C03295=1188.011,290.070,-68.548,-176.804,7.489,148.492
C03296=1188.007,290.318,-68.578,-176.802,7.491,148.492
C03297=1188.002,290.566,-68.607,-176.799,7.494,148.492
C03298=1187.998,290.815,-68.636,-176.796,7.497,148.492
C03299=1187.994,291.063,-68.665,-176.794,7.500,148.492
C03300=1187.990,291.311,-68.695,-176.791,7.502,148.492
C03301=1187.985,291.559,-68.724,-176.789,7.505,148.492
C03302=1187.980,291.808,-68.754,-176.786,7.508,148.492
C03303=1187.976,292.056,-68.784,-176.783,7.511,148.492
C03304=1187.972,292.305,-68.813,-176.781,7.514,148.492
C03305=1187.968,292.553,-68.843,-176.778,7.517,148.492
C03306=1187.964,292.801,-68.872,-176.776,7.520,148.492
C03307=1187.959,293.049,-68.901,-176.773,7.523,148.492
C03308=1187.955,293.297,-68.931,-176.771,7.525,148.492
C03309=1187.951,293.545,-68.961,-176.768,7.528,148.492
C03310=1187.947,293.793,-68.990,-176.765,7.531,148.492
C03311=1187.943,294.041,-69.020,-176.763,7.534,148.491
C03312=1187.938,294.289,-69.049,-176.761,7.536,148.491
C03313=1187.933,294.538,-69.079,-176.758,7.539,148.492
C03314=1187.929,294.786,-69.109,-176.756,7.542,148.492
C03315=1187.925,295.035,-69.138,-176.753,7.545,148.492
C03316=1187.921,295.283,-69.167,-176.751,7.547,148.491
C03317=1187.917,295.531,-69.197,-176.748,7.550,148.491
C03318=1187.913,295.779,-69.227,-176.745,7.553,148.491
C03319=1187.908,296.027,-69.257,-176.743,7.556,148.491
C03320=1187.904,296.276,-69.287,-176.740,7.559,148.491
C03321=1187.900,296.524,-69.316,-176.738,7.562,148.491
C03322=1187.896,296.771,-69.346,-176.735,7.565,148.491
C03323=1187.891,297.020,-69.376,-176.732,7.568,148.491
C03324=1187.887,297.268,-69.406,-176.730,7.570,148.491
C03325=1187.882,297.517,-69.435,-176.727,7.573,148.491
C03326=1187.878,297.764,-69.465,-176.725,7.576,148.491
C03327=1187.874,298.012,-69.495,-176.722,7.579,148.491
C03328=1187.869,298.261,-69.525,-176.720,7.581,148.491
C03329=1187.866,298.509,-69.555,-176.718,7.584,148.491
C03330=1187.861,298.757,-69.584,-176.715,7.587,148.491
C03331=1187.856,299.006,-69.615,-176.712,7.590,148.491
C03332=1187.853,299.253,-69.645,-176.709,7.593,148.491
C03333=1187.848,299.501,-69.674,-176.707,7.595,148.491
C03334=1187.843,299.750,-69.704,-176.705,7.598,148.491
C03335=1187.840,299.998,-69.734,-176.702,7.602,148.491
C03336=1187.835,300.246,-69.764,-176.700,7.605,148.491
C03337=1187.831,300.494,-69.795,-176.698,7.607,148.491
C03338=1187.827,300.743,-69.824,-176.695,7.610,148.491
C03339=1187.823,300.991,-69.854,-176.692,7.613,148.491
C03340=1187.818,301.239,-69.885,-176.689,7.616,148.491
C03341=1187.814,301.487,-69.914,-176.687,7.619,148.491
C03342=1187.810,301.735,-69.944,-176.685,7.621,148.491
C03343=1187.805,301.984,-69.974,-176.682,7.624,148.491
C03344=1187.802,302.231,-70.004,-176.680,7.627,148.491
C03345=1187.797,302.480,-70.034,-176.677,7.630,148.491
C03346=1187.793,302.727,-70.065,-176.674,7.633,148.491
C03347=1187.788,302.976,-70.095,-176.672,7.636,148.491
C03348=1187.784,303.224,-70.125,-176.669,7.639,148.491
C03349=1187.781,303.472,-70.155,-176.667,7.642,148.491
C03350=1187.776,303.721,-70.185,-176.664,7.645,148.491
C03351=1187.772,303.968,-70.216,-176.662,7.648,148.491
C03352=1187.767,304.217,-70.246,-176.659,7.650,148.491
C03353=1187.763,304.465,-70.276,-176.657,7.653,148.491
C03354=1187.758,304.712,-70.307,-176.654,7.656,148.491
C03355=1187.754,304.961,-70.336,-176.652,7.659,148.491
C03356=1187.750,305.209,-70.367,-176.649,7.662,148.491
C03357=1187.746,305.457,-70.397,-176.647,7.665,148.491
C03358=1187.741,305.706,-70.427,-176.644,7.668,148.491
C03359=1187.738,305.953,-70.458,-176.641,7.671,148.491
C03360=1187.733,306.201,-70.488,-176.639,7.674,148.491
C03361=1187.728,306.449,-70.519,-176.637,7.677,148.491
C03362=1187.725,306.698,-70.549,-176.634,7.679,148.491
C03363=1187.720,306.946,-70.580,-176.632,7.682,148.491
C03364=1187.716,307.194,-70.610,-176.629,7.685,148.491
C03365=1187.712,307.442,-70.641,-176.627,7.688,148.492
C03366=1187.708,307.690,-70.670,-176.624,7.691,148.492
C03367=1187.704,307.939,-70.701,-176.622,7.694,148.491
C03368=1187.699,308.187,-70.732,-176.619,7.697,148.491
C03369=1187.695,308.434,-70.762,-176.617,7.700,148.492
C03370=1187.690,308.682,-70.793,-176.614,7.703,148.492
C03371=1187.686,308.931,-70.824,-176.611,7.706,148.492
C03372=1187.682,309.179,-70.853,-176.609,7.708,148.492
C03373=1187.678,309.427,-70.884,-176.607,7.711,148.492
C03374=1187.674,309.675,-70.914,-176.604,7.714,148.492
C03375=1187.670,309.923,-70.946,-176.602,7.717,148.492
C03376=1187.665,310.171,-70.976,-176.599,7.720,148.492
C03377=1187.661,310.419,-71.006,-176.596,7.723,148.492
C03378=1187.657,310.667,-71.037,-176.595,7.726,148.492
C03379=1187.653,310.916,-71.068,-176.592,7.729,148.492
C03380=1187.648,311.164,-71.099,-176.589,7.732,148.492
C03381=1187.644,311.411,-71.129,-176.587,7.735,148.492
C03382=1187.639,311.659,-71.160,-176.584,7.738,148.492
C03383=1187.635,311.908,-71.191,-176.581,7.741,148.492
C03384=1187.632,312.155,-71.221,-176.579,7.743,148.492
C03385=1187.627,312.403,-71.252,-176.577,7.747,148.492
C03386=1187.623,312.652,-71.283,-176.574,7.750,148.492
C03387=1187.618,312.900,-71.314,-176.572,7.753,148.492
C03388=1187.614,313.148,-71.344,-176.569,7.756,148.492
C03389=1187.610,313.396,-71.375,-176.567,7.759,148.492
C03390=1187.606,313.644,-71.406,-176.565,7.761,148.492
C03391=1187.601,313.892,-71.437,-176.562,7.764,148.492
C03392=1187.597,314.169,-71.471,-176.559,7.768,148.492
C03393=1187.593,314.445,-71.506,-176.556,7.771,148.492
C03394=1187.587,314.722,-71.540,-176.554,7.774,148.492
C03395=1187.583,314.999,-71.575,-176.551,7.777,148.492
C03396=1187.578,315.246,-71.606,-176.549,7.781,148.493
C03397=1187.575,315.495,-71.638,-176.546,7.784,148.493
C03398=1187.571,315.742,-71.668,-176.543,7.787,148.493
C03399=1187.566,315.990,-71.698,-176.541,7.790,148.493
C03400=1187.562,316.239,-71.730,-176.538,7.793,148.493
C03401=1187.557,316.487,-71.760,-176.536,7.795,148.493
C03402=1187.553,316.734,-71.792,-176.534,7.799,148.493
C03403=1187.549,316.983,-71.823,-176.531,7.802,148.493
C03404=1187.545,317.231,-71.854,-176.528,7.805,148.493
C03405=1187.541,317.479,-71.886,-176.526,7.808,148.493
C03406=1187.536,317.727,-71.916,-176.523,7.811,148.493
C03407=1187.533,317.975,-71.947,-176.521,7.814,148.493
C03408=1187.529,318.222,-71.978,-176.519,7.816,148.493
C03409=1187.524,318.470,-72.009,-176.516,7.819,148.493
C03410=1187.520,318.719,-72.040,-176.514,7.823,148.494
C03411=1187.516,318.966,-72.072,-176.511,7.826,148.493
C03412=1187.512,319.215,-72.103,-176.509,7.829,148.493
C03413=1187.507,319.462,-72.134,-176.506,7.832,148.494
C03414=1187.503,319.711,-72.165,-176.504,7.835,148.494
C03415=1187.499,319.959,-72.196,-176.502,7.838,148.494
C03416=1187.495,320.207,-72.228,-176.499,7.841,148.494
C03417=1187.490,320.455,-72.259,-176.497,7.844,148.494
C03418=1187.487,320.703,-72.291,-176.494,7.847,148.494
C03419=1187.482,320.951,-72.321,-176.492,7.850,148.494
C03420=1187.478,321.199,-72.353,-176.489,7.853,148.494
C03421=1187.474,321.447,-72.384,-176.487,7.856,148.494
C03422=1187.470,321.695,-72.416,-176.485,7.858,148.494
C03423=1187.465,321.943,-72.447,-176.482,7.862,148.494
C03424=1187.462,322.191,-72.479,-176.480,7.865,148.494
C03425=1187.457,322.438,-72.510,-176.477,7.868,148.495
C03426=1187.453,322.687,-72.542,-176.475,7.871,148.495
C03427=1187.448,322.935,-72.573,-176.472,7.874,148.495
C03428=1187.444,323.183,-72.604,-176.470,7.877,148.495
C03429=1187.440,323.431,-72.636,-176.467,7.881,148.495
C03430=1187.436,323.679,-72.668,-176.465,7.883,148.495
C03431=1187.432,323.927,-72.698,-176.463,7.886,148.495
C03432=1187.428,324.175,-72.730,-176.460,7.889,148.495
C03433=1187.424,324.422,-72.762,-176.458,7.892,148.495
C03434=1187.420,324.671,-72.793,-176.455,7.896,148.495
C03435=1187.415,324.918,-72.825,-176.453,7.899,148.495
C03436=1187.411,325.166,-72.857,-176.450,7.902,148.496
C03437=1187.407,325.415,-72.888,-176.448,7.905,148.496
C03438=1187.403,325.662,-72.919,-176.446,7.907,148.496
C03439=1187.399,325.910,-72.951,-176.443,7.910,148.496
C03440=1187.395,326.158,-72.983,-176.441,7.914,148.496
C03441=1187.390,326.407,-73.014,-176.438,7.917,148.496
C03442=1187.386,326.655,-73.046,-176.436,7.920,148.496
C03443=1187.382,326.902,-73.078,-176.433,7.923,148.496
C03444=1187.378,327.150,-73.110,-176.431,7.926,148.496
C03445=1187.373,327.398,-73.142,-176.429,7.930,148.497
C03446=1187.369,327.646,-73.173,-176.426,7.933,148.497
C03447=1187.365,327.894,-73.205,-176.425,7.935,148.497
C03448=1187.361,328.142,-73.236,-176.422,7.938,148.497
C03449=1187.357,328.390,-73.269,-176.420,7.942,148.497
C03450=1187.352,328.637,-73.300,-176.417,7.945,148.497
C03451=1187.349,328.885,-73.332,-176.415,7.948,148.497
C03452=1187.345,329.134,-73.364,-176.412,7.951,148.497
C03453=1187.340,329.381,-73.396,-176.410,7.954,148.497
C03454=1187.336,329.629,-73.428,-176.407,7.958,148.498
C03455=1187.332,329.877,-73.460,-176.405,7.961,148.498
C03456=1187.327,330.126,-73.491,-176.403,7.963,148.498
C03457=1187.323,330.374,-73.523,-176.400,7.966,148.498
C03458=1187.320,330.622,-73.555,-176.398,7.969,148.498
C03459=1187.315,330.869,-73.587,-176.396,7.973,148.498
C03460=1187.311,331.117,-73.619,-176.393,7.976,148.498
C03461=1187.307,331.366,-73.651,-176.391,7.979,148.498
C03462=1187.303,331.612,-73.683,-176.388,7.982,148.498
C03463=1187.299,331.860,-73.715,-176.386,7.985,148.499
C03464=1187.294,332.109,-73.747,-176.384,7.989,148.499
C03465=1187.290,332.356,-73.779,-176.382,7.991,148.499
C03466=1187.286,332.604,-73.811,-176.379,7.994,148.499
C03467=1187.282,332.852,-73.843,-176.377,7.997,148.499
C03468=1187.278,333.101,-73.875,-176.374,8.000,148.499
C03469=1187.273,333.348,-73.907,-176.372,8.004,148.499
C03470=1187.269,333.596,-73.939,-176.370,8.007,148.500
C03471=1187.265,333.845,-73.971,-176.367,8.010,148.500
C03472=1187.262,334.092,-74.004,-176.365,8.013,148.500
C03473=1187.257,334.340,-74.036,-176.363,8.017,148.500
C03474=1187.253,334.588,-74.068,-176.360,8.020,148.500
C03475=1187.248,334.836,-74.100,-176.358,8.022,148.500
C03476=1187.245,335.084,-74.132,-176.356,8.026,148.500
C03477=1187.240,335.331,-74.165,-176.353,8.029,148.500
C03478=1187.236,335.579,-74.197,-176.351,8.032,148.501
C03479=1187.232,335.827,-74.229,-176.349,8.035,148.501
C03480=1187.228,336.076,-74.261,-176.347,8.039,148.501
C03481=1187.223,336.323,-74.294,-176.344,8.042,148.501
C03482=1187.220,336.571,-74.326,-176.342,8.045,148.501
C03483=1187.215,336.819,-74.358,-176.339,8.048,148.501
C03484=1187.212,337.066,-74.391,-176.337,8.052,148.502
C03485=1187.207,337.315,-74.423,-176.334,8.055,148.502
C03486=1187.203,337.562,-74.455,-176.333,8.057,148.502
C03487=1187.199,337.810,-74.488,-176.330,8.060,148.502
C03488=1187.194,338.058,-74.520,-176.328,8.064,148.502
C03489=1187.191,338.306,-74.553,-176.325,8.067,148.502
C03490=1187.187,338.554,-74.585,-176.323,8.070,148.502
C03491=1187.182,338.801,-74.617,-176.321,8.073,148.503
C03492=1187.178,339.049,-74.650,-176.319,8.077,148.503
C03493=1187.174,339.297,-74.682,-176.316,8.080,148.503
C03494=1187.170,339.545,-74.715,-176.314,8.083,148.503
C03495=1187.166,339.793,-74.747,-176.312,8.086,148.503
C03496=1187.161,340.072,-74.784,-176.309,8.090,148.504
C03497=1187.157,340.350,-74.820,-176.306,8.094,148.504
C03498=1187.152,340.629,-74.858,-176.304,8.097,148.504
C03499=1187.147,340.908,-74.893,-176.302,8.100,148.504
C03500=1187.143,341.156,-74.927,-176.299,8.103,148.504
C03501=1187.139,341.404,-74.958,-176.297,8.107,148.504
C03502=1187.135,341.652,-74.992,-176.295,8.110,148.505
C03503=1187.131,341.899,-75.025,-176.292,8.113,148.505
C03504=1187.127,342.147,-75.057,-176.290,8.117,148.505
C03505=1187.122,342.395,-75.089,-176.288,8.120,148.505
C03506=1187.118,342.643,-75.122,-176.286,8.123,148.506
C03507=1187.114,342.891,-75.155,-176.283,8.127,148.506
C03508=1187.110,343.138,-75.188,-176.281,8.130,148.506
C03509=1187.106,343.386,-75.220,-176.279,8.133,148.506
C03510=1187.102,343.634,-75.253,-176.277,8.135,148.506
C03511=1187.098,343.882,-75.286,-176.275,8.139,148.506
C03512=1187.093,344.130,-75.319,-176.272,8.142,148.507
C03513=1187.090,344.378,-75.351,-176.270,8.145,148.507
C03514=1187.086,344.625,-75.384,-176.268,8.149,148.507
C03515=1187.081,344.874,-75.417,-176.266,8.152,148.507
C03516=1187.077,345.121,-75.450,-176.263,8.155,148.507
C03517=1187.073,345.369,-75.483,-176.261,8.159,148.508
C03518=1187.068,345.616,-75.516,-176.259,8.162,148.508
C03519=1187.065,345.864,-75.548,-176.257,8.165,148.508
C03520=1187.060,346.112,-75.581,-176.254,8.169,148.508
C03521=1187.056,346.360,-75.614,-176.252,8.172,148.509
C03522=1187.052,346.607,-75.647,-176.250,8.175,148.509
C03523=1187.048,346.855,-75.680,-176.248,8.179,148.509
C03524=1187.044,347.103,-75.714,-176.246,8.181,148.509
C03525=1187.039,347.351,-75.746,-176.244,8.184,148.509
C03526=1187.035,347.599,-75.779,-176.241,8.188,148.510
C03527=1187.031,347.847,-75.812,-176.239,8.191,148.510
C03528=1187.028,348.094,-75.845,-176.237,8.195,148.510
C03529=1187.024,348.342,-75.878,-176.235,8.198,148.511
C03530=1187.020,348.590,-75.911,-176.233,8.201,148.511
C03531=1187.015,348.837,-75.944,-176.231,8.205,148.511
C03532=1187.011,349.085,-75.978,-176.228,8.208,148.511
C03533=1187.007,349.333,-76.011,-176.226,8.211,148.511
C03534=1187.003,349.580,-76.044,-176.224,8.215,148.512
C03535=1186.999,349.828,-76.077,-176.222,8.218,148.512
C03536=1186.995,350.077,-76.111,-176.219,8.221,148.512
C03537=1186.991,350.324,-76.144,-176.218,8.225,148.512
C03538=1186.987,350.572,-76.177,-176.215,8.228,148.513
C03539=1186.983,350.820,-76.210,-176.214,8.231,148.513
C03540=1186.979,351.068,-76.243,-176.211,8.234,148.513
C03541=1186.975,351.315,-76.276,-176.209,8.237,148.513
C03542=1186.970,351.563,-76.310,-176.207,8.241,148.514
C03543=1186.966,351.811,-76.343,-176.205,8.244,148.514
C03544=1186.962,352.058,-76.376,-176.203,8.248,148.514
C03545=1186.958,352.306,-76.409,-176.201,8.251,148.514
C03546=1186.954,352.554,-76.442,-176.198,8.254,148.515
C03547=1186.950,352.802,-76.475,-176.196,8.258,148.515
C03548=1186.946,353.049,-76.509,-176.194,8.261,148.515
C03549=1186.942,353.297,-76.543,-176.192,8.265,148.516
C03550=1186.938,353.545,-76.576,-176.190,8.268,148.516
C03551=1186.933,353.793,-76.610,-176.188,8.272,148.516
C03552=1186.929,354.041,-76.643,-176.186,8.275,148.516
C03553=1186.925,354.288,-76.676,-176.183,8.278,148.517
C03554=1186.921,354.535,-76.710,-176.182,8.282,148.517
C03555=1186.917,354.783,-76.743,-176.179,8.285,148.517
C03556=1186.913,355.031,-76.776,-176.178,8.288,148.517
C03557=1186.909,355.279,-76.810,-176.175,8.291,148.518
C03558=1186.905,355.527,-76.844,-176.174,8.295,148.518
C03559=1186.901,355.775,-76.877,-176.171,8.298,148.518
C03560=1186.897,356.022,-76.910,-176.170,8.301,148.519
C03561=1186.893,356.269,-76.944,-176.167,8.305,148.519
C03562=1186.889,356.517,-76.977,-176.165,8.308,148.519
C03563=1186.885,356.766,-77.011,-176.163,8.312,148.520
C03564=1186.881,357.013,-77.045,-176.161,8.315,148.520
C03565=1186.876,357.261,-77.079,-176.159,8.319,148.520
C03566=1186.872,357.508,-77.112,-176.157,8.322,148.521
C03567=1186.868,357.756,-77.146,-176.155,8.325,148.521
C03568=1186.865,358.004,-77.179,-176.153,8.329,148.521
C03569=1186.860,358.252,-77.213,-176.151,8.332,148.521
C03570=1186.856,358.499,-77.247,-176.149,8.336,148.522
C03571=1186.852,358.747,-77.280,-176.147,8.339,148.522
C03572=1186.848,358.994,-77.314,-176.145,8.343,148.522
C03573=1186.844,359.243,-77.348,-176.143,8.345,148.523
C03574=1186.840,359.490,-77.382,-176.141,8.349,148.523
C03575=1186.836,359.738,-77.415,-176.139,8.352,148.523
C03576=1186.831,359.985,-77.449,-176.137,8.356,148.524
C03577=1186.828,360.233,-77.483,-176.135,8.360,148.524
C03578=1186.824,360.480,-77.517,-176.133,8.363,148.524
C03579=1186.820,360.728,-77.550,-176.131,8.366,148.525
C03580=1186.815,360.976,-77.584,-176.129,8.370,148.525
C03581=1186.812,361.224,-77.618,-176.127,8.373,148.526
C03582=1186.808,361.471,-77.652,-176.126,8.377,148.526
C03583=1186.803,361.719,-77.686,-176.124,8.380,148.526
C03584=1186.799,361.966,-77.719,-176.122,8.383,148.527
C03585=1186.796,362.214,-77.754,-176.120,8.387,148.527
C03586=1186.791,362.462,-77.787,-176.118,8.390,148.527
C03587=1186.787,362.709,-77.821,-176.116,8.394,148.528
C03588=1186.783,362.957,-77.856,-176.114,8.397,148.528
C03589=1186.779,363.205,-77.889,-176.113,8.400,148.528
C03590=1186.775,363.452,-77.923,-176.111,8.403,148.529
C03591=1186.771,363.700,-77.958,-176.109,8.407,148.529
C03592=1186.767,363.948,-77.991,-176.107,8.411,148.530
C03593=1186.763,364.195,-78.025,-176.105,8.414,148.530
C03594=1186.759,364.443,-78.059,-176.104,8.418,148.530
C03595=1186.755,364.691,-78.093,-176.102,8.421,148.531
C03596=1186.751,364.938,-78.127,-176.100,8.424,148.531
C03597=1186.748,365.186,-78.162,-176.098,8.428,148.531
C03598=1186.743,365.434,-78.196,-176.097,8.431,148.532
C03599=1186.739,365.681,-78.229,-176.095,8.434,148.532
C03600=1186.735,365.963,-78.268,-176.093,8.439,148.533
C03601=1186.730,366.244,-78.308,-176.091,8.442,148.533
C03602=1186.725,366.525,-78.346,-176.089,8.446,148.534
C03603=1186.721,366.806,-78.385,-176.087,8.450,148.534
C03604=1186.716,367.054,-78.419,-176.086,8.453,148.534
C03605=1186.713,367.302,-78.453,-176.084,8.457,148.535
C03606=1186.708,367.550,-78.487,-176.083,8.461,148.536
C03607=1186.704,367.797,-78.521,-176.081,8.463,148.536
C03608=1186.700,368.045,-78.556,-176.079,8.467,148.536
C03609=1186.697,368.292,-78.590,-176.078,8.471,148.537
C03610=1186.693,368.540,-78.625,-176.076,8.474,148.537
C03611=1186.689,368.787,-78.659,-176.075,8.477,148.538
C03612=1186.684,369.035,-78.693,-176.073,8.481,148.538
C03613=1186.681,369.282,-78.727,-176.071,8.484,148.539
C03614=1186.676,369.530,-78.761,-176.070,8.487,148.539
C03615=1186.672,369.779,-78.796,-176.068,8.491,148.539
C03616=1186.668,370.026,-78.830,-176.067,8.494,148.540
C03617=1186.664,370.273,-78.864,-176.065,8.498,148.540
C03618=1186.661,370.521,-78.899,-176.064,8.501,148.541
C03619=1186.656,370.768,-78.933,-176.062,8.504,148.541
C03620=1186.652,371.016,-78.968,-176.061,8.508,148.542
C03621=1186.648,371.264,-79.002,-176.059,8.511,148.542
C03622=1186.644,371.512,-79.037,-176.058,8.514,148.543
C03623=1186.640,371.759,-79.070,-176.056,8.518,148.543
C03624=1186.636,372.006,-79.105,-176.055,8.521,148.544
C03625=1186.632,372.254,-79.140,-176.053,8.525,148.544
C03626=1186.628,372.501,-79.174,-176.052,8.527,148.544
C03627=1186.624,372.749,-79.209,-176.051,8.531,148.545
C03628=1186.620,372.996,-79.244,-176.050,8.534,148.545
C03629=1186.617,373.244,-79.278,-176.048,8.538,148.546
C03630=1186.612,373.492,-79.312,-176.047,8.541,148.546
C03631=1186.608,373.740,-79.347,-176.045,8.544,148.547
C03632=1186.604,373.987,-79.381,-176.044,8.548,148.548
C03633=1186.600,374.235,-79.416,-176.043,8.551,148.548
C03634=1186.596,374.482,-79.451,-176.042,8.554,148.549
C03635=1186.593,374.730,-79.485,-176.040,8.558,148.549
C03636=1186.588,374.977,-79.520,-176.039,8.561,148.550
C03637=1186.584,375.225,-79.555,-176.037,8.565,148.550
C03638=1186.580,375.472,-79.589,-176.037,8.568,148.551
C03639=1186.576,375.720,-79.623,-176.035,8.571,148.551
C03640=1186.572,375.967,-79.658,-176.034,8.574,148.552
C03641=1186.568,376.215,-79.693,-176.033,8.577,148.552
C03642=1186.564,376.463,-79.728,-176.031,8.581,148.553
C03643=1186.560,376.710,-79.762,-176.030,8.584,148.553
C03644=1186.556,376.957,-79.797,-176.029,8.588,148.554
C03645=1186.552,377.205,-79.832,-176.028,8.591,148.554
C03646=1186.548,377.453,-79.866,-176.027,8.594,148.555
C03647=1186.544,377.701,-79.901,-176.025,8.598,148.555
C03648=1186.540,377.947,-79.936,-176.024,8.601,148.556
C03649=1186.536,378.196,-79.971,-176.023,8.604,148.556
C03650=1186.532,378.443,-80.005,-176.022,8.607,148.557
C03651=1186.528,378.690,-80.041,-176.021,8.611,148.557
C03652=1186.524,378.938,-80.075,-176.020,8.613,148.558
C03653=1186.520,379.186,-80.109,-176.019,8.617,148.558
C03654=1186.516,379.432,-80.145,-176.018,8.620,148.559
C03655=1186.512,379.681,-80.179,-176.017,8.624,148.560
C03656=1186.508,379.929,-80.214,-176.016,8.627,148.560
